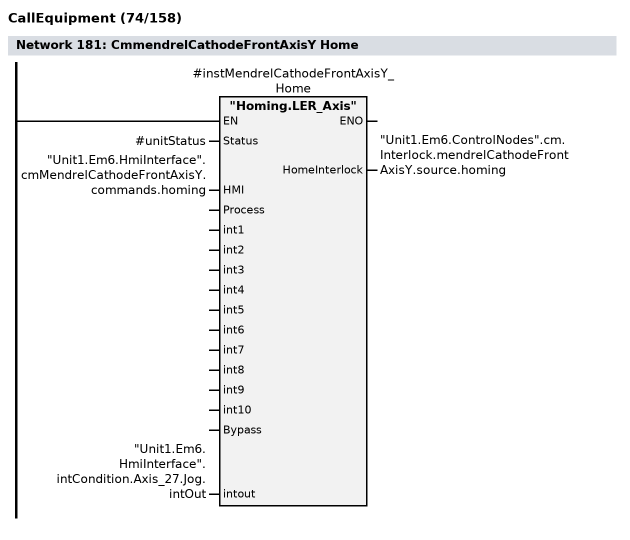
   RUNG wire#powerrail
      #instMendrelCathodeFrontAxisY_Home(Status := #unitStatus, HMI := "Unit1.Em6.HmiInterface".cmMendrelCathodeFrontAxisY.commands.homing, Process :=, int1 :=, int2 :=, int3 :=, int4 :=, int5 :=, int6 :=, int7 :=, int8 :=, int9 :=, int10 :=, Bypass :=, intout := "Unit1.Em6.HmiInterface".intCondition.Axis_27.Jog.intOut, HomeInterlock => "Unit1.Em6.ControlNodes".cm.Interlock.mendrelCathodeFrontAxisY.source.homing)
   END_RUNG
   // the same network as SCL:
   #instMendrelCathodeFrontAxisY_Home(Status := #unitStatus,   // "Homing.LER_Axis"
                           HMI := "Unit1.Em6.HmiInterface".cmMendrelCathodeFrontAxisY.commands.homing,
                           intout := "Unit1.Em6.HmiInterface".intCondition.Axis_27.Jog.intOut,
                           HomeInterlock => "Unit1.Em6.ControlNodes".cm.Interlock.mendrelCathodeFrontAxisY.source.homing);
END_REGION

REGION Network 182: CmMendrelCathodeFrontAxisY Position Absolute Jog
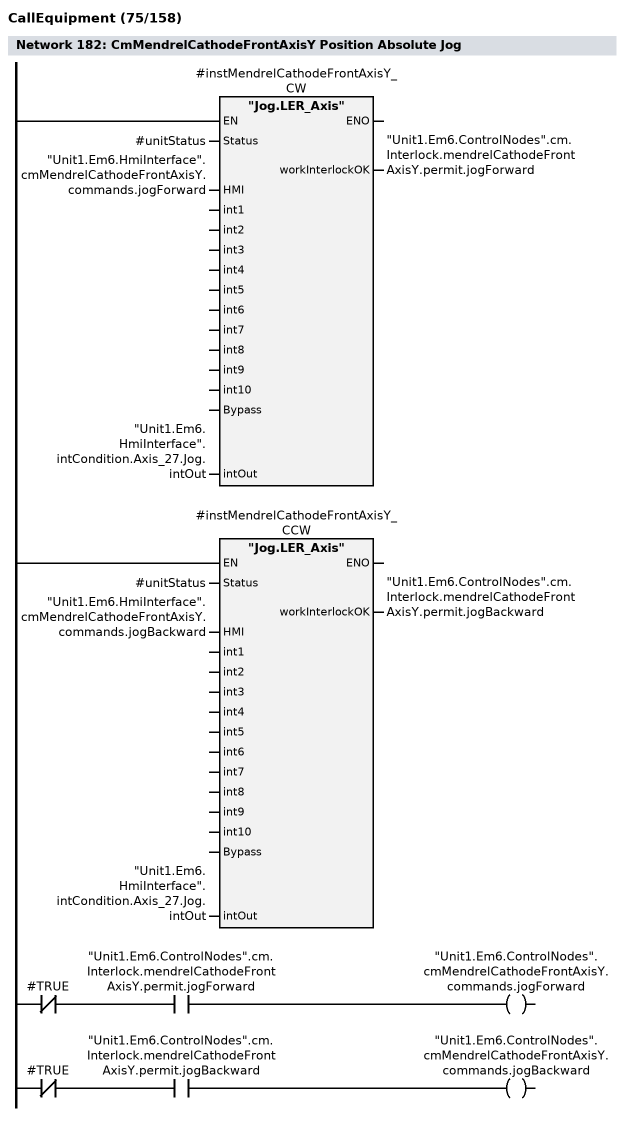
   RUNG wire#powerrail
      #instMendrelCathodeFrontAxisY_CW(Status := #unitStatus, HMI := "Unit1.Em6.HmiInterface".cmMendrelCathodeFrontAxisY.commands.jogForward, int1 :=, int2 :=, int3 :=, int4 :=, int5 :=, int6 :=, int7 :=, int8 :=, int9 :=, int10 :=, Bypass :=, intOut := "Unit1.Em6.HmiInterface".intCondition.Axis_27.Jog.intOut, workInterlockOK => "Unit1.Em6.ControlNodes".cm.Interlock.mendrelCathodeFrontAxisY.permit.jogForward)
   END_RUNG
   RUNG wire#powerrail
      #instMendrelCathodeFrontAxisY_CCW(Status := #unitStatus, HMI := "Unit1.Em6.HmiInterface".cmMendrelCathodeFrontAxisY.commands.jogBackward, int1 :=, int2 :=, int3 :=, int4 :=, int5 :=, int6 :=, int7 :=, int8 :=, int9 :=, int10 :=, Bypass :=, intOut := "Unit1.Em6.HmiInterface".intCondition.Axis_27.Jog.intOut, workInterlockOK => "Unit1.Em6.ControlNodes".cm.Interlock.mendrelCathodeFrontAxisY.permit.jogBackward)
   END_RUNG
   RUNG wire#powerrail
      I_Contact( #TRUE )
      Contact( "Unit1.Em6.ControlNodes".cm.Interlock.mendrelCathodeFrontAxisY.permit.jogForward )
      Coil( "Unit1.Em6.ControlNodes".cmMendrelCathodeFrontAxisY.commands.jogForward )
   END_RUNG
   RUNG wire#powerrail
      I_Contact( #TRUE )
      Contact( "Unit1.Em6.ControlNodes".cm.Interlock.mendrelCathodeFrontAxisY.permit.jogBackward )
      Coil( "Unit1.Em6.ControlNodes".cmMendrelCathodeFrontAxisY.commands.jogBackward )
   END_RUNG
   // the same network as SCL:
   #instMendrelCathodeFrontAxisY_CW(Status := #unitStatus,   // "Jog.LER_Axis"
                           HMI := "Unit1.Em6.HmiInterface".cmMendrelCathodeFrontAxisY.commands.jogForward,
                           intOut := "Unit1.Em6.HmiInterface".intCondition.Axis_27.Jog.intOut,
                           workInterlockOK => "Unit1.Em6.ControlNodes".cm.Interlock.mendrelCathodeFrontAxisY.permit.jogForward);
   #instMendrelCathodeFrontAxisY_CCW(Status := #unitStatus,   // "Jog.LER_Axis"
                           HMI := "Unit1.Em6.HmiInterface".cmMendrelCathodeFrontAxisY.commands.jogBackward,
                           intOut := "Unit1.Em6.HmiInterface".intCondition.Axis_27.Jog.intOut,
                           workInterlockOK => "Unit1.Em6.ControlNodes".cm.Interlock.mendrelCathodeFrontAxisY.permit.jogBackward);
   "Unit1.Em6.ControlNodes".cmMendrelCathodeFrontAxisY.commands.jogForward := NOT #TRUE AND "Unit1.Em6.ControlNodes".cm.Interlock.mendrelCathodeFrontAxisY.permit.jogForward;
   "Unit1.Em6.ControlNodes".cmMendrelCathodeFrontAxisY.commands.jogBackward := NOT #TRUE AND "Unit1.Em6.ControlNodes".cm.Interlock.mendrelCathodeFrontAxisY.permit.jogBackward;
END_REGION

REGION Network 183: CmMendrelCathodeFrontAxisY Position Absolute Position0
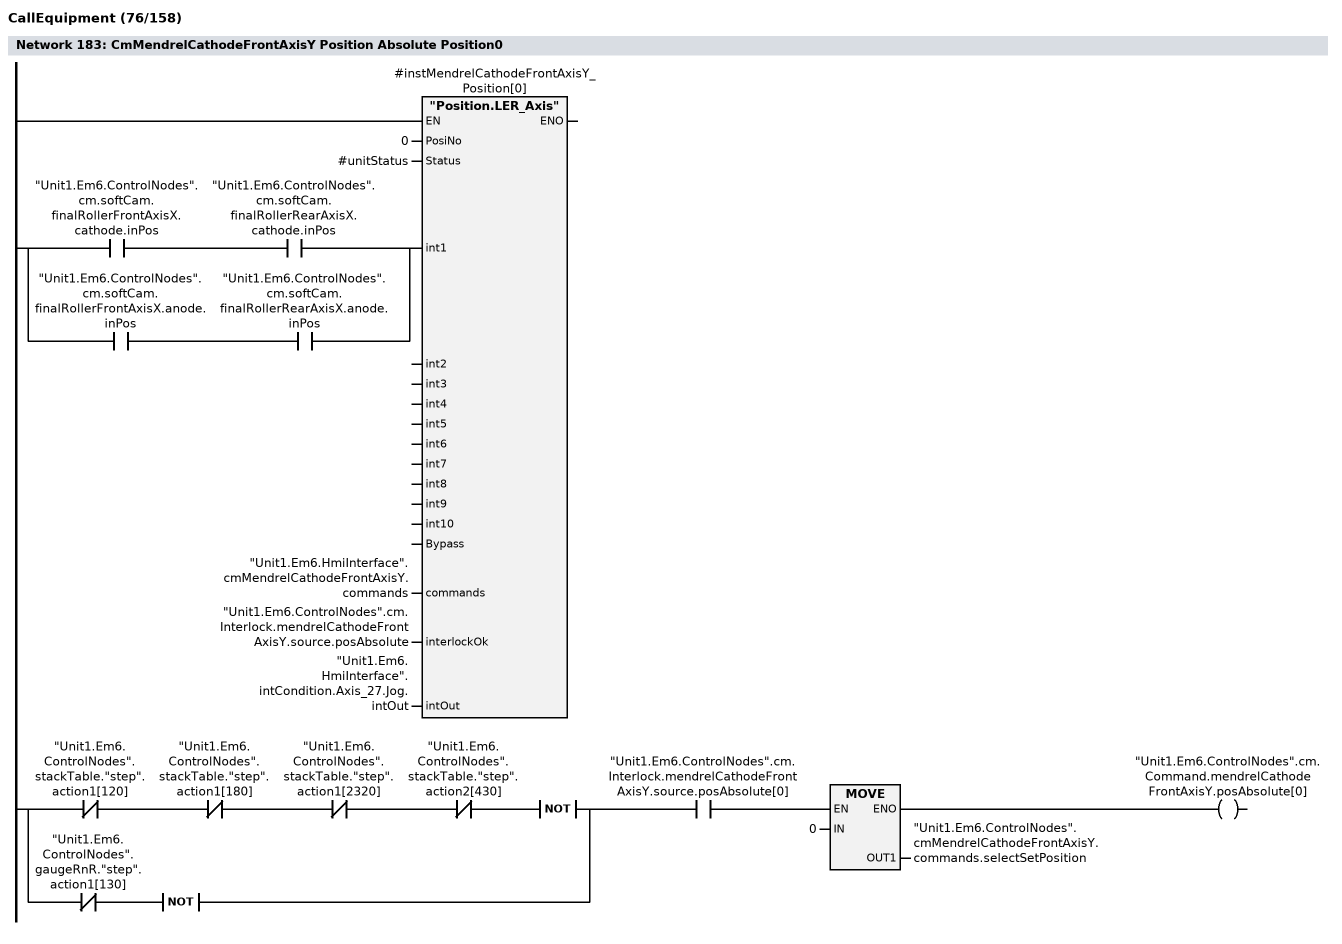
   RUNG wire#powerrail
      #instMendrelCathodeFrontAxisY_Position[0](int1 := wire#w1, PosiNo := 0, Status := #unitStatus, int2 :=, int3 :=, int4 :=, int5 :=, int6 :=, int7 :=, int8 :=, int9 :=, int10 :=, Bypass :=, commands := "Unit1.Em6.HmiInterface".cmMendrelCathodeFrontAxisY.commands, interlockOk := "Unit1.Em6.ControlNodes".cm.Interlock.mendrelCathodeFrontAxisY.source.posAbsolute, intOut := "Unit1.Em6.HmiInterface".intCondition.Axis_27.Jog.intOut)
   END_RUNG
   RUNG wire#powerrail
      Contact( "Unit1.Em6.ControlNodes".cm.softCam.finalRollerFrontAxisX.cathode.inPos )
      Contact( "Unit1.Em6.ControlNodes".cm.softCam.finalRollerRearAxisX.cathode.inPos )
   END_RUNG wire#w1
   RUNG wire#powerrail
      Contact( "Unit1.Em6.ControlNodes".cm.softCam.finalRollerFrontAxisX.anode.inPos )
      Contact( "Unit1.Em6.ControlNodes".cm.softCam.finalRollerRearAxisX.anode.inPos )
   END_RUNG wire#w1
   RUNG wire#powerrail
      I_Contact( "Unit1.Em6.ControlNodes".stackTable."step".action1[120] )
      I_Contact( "Unit1.Em6.ControlNodes".stackTable."step".action1[180] )
      I_Contact( "Unit1.Em6.ControlNodes".stackTable."step".action1[2320] )
      I_Contact( "Unit1.Em6.ControlNodes".stackTable."step".action2[430] )
      Not()
      wire#w2
      Contact( "Unit1.Em6.ControlNodes".cm.Interlock.mendrelCathodeFrontAxisY.source.posAbsolute[0] )
      Move(in := 0, out1 => "Unit1.Em6.ControlNodes".cmMendrelCathodeFrontAxisY.commands.selectSetPosition)
      Coil( "Unit1.Em6.ControlNodes".cm.Command.mendrelCathodeFrontAxisY.posAbsolute[0] )
   END_RUNG
   RUNG wire#powerrail
      I_Contact( "Unit1.Em6.ControlNodes".gaugeRnR."step".action1[130] )
      Not()
   END_RUNG wire#w2
   // the same network as SCL:
   #instMendrelCathodeFrontAxisY_Position[0](PosiNo := 0,   // "Position.LER_Axis"
                           Status := #unitStatus,
                           int1 := ("Unit1.Em6.ControlNodes".cm.softCam.finalRollerFrontAxisX.cathode.inPos AND "Unit1.Em6.ControlNodes".cm.softCam.finalRollerRearAxisX.cathode.inPos) OR ("Unit1.Em6.ControlNodes".cm.softCam.finalRollerFrontAxisX.anode.inPos AND "Unit1.Em6.ControlNodes".cm.softCam.finalRollerRearAxisX.anode.inPos),
                           commands := "Unit1.Em6.HmiInterface".cmMendrelCathodeFrontAxisY.commands,
                           interlockOk := "Unit1.Em6.ControlNodes".cm.Interlock.mendrelCathodeFrontAxisY.source.posAbsolute,
                           intOut := "Unit1.Em6.HmiInterface".intCondition.Axis_27.Jog.intOut);
   #_w1 := (NOT (NOT "Unit1.Em6.ControlNodes".stackTable."step".action1[120] AND NOT "Unit1.Em6.ControlNodes".stackTable."step".action1[180] AND NOT "Unit1.Em6.ControlNodes".stackTable."step".action1[2320] AND NOT "Unit1.Em6.ControlNodes".stackTable."step".action2[430]) OR NOT (NOT "Unit1.Em6.ControlNodes".gaugeRnR."step".action1[130])) AND "Unit1.Em6.ControlNodes".cm.Interlock.mendrelCathodeFrontAxisY.source.posAbsolute[0];
   IF #_w1 THEN "Unit1.Em6.ControlNodes".cmMendrelCathodeFrontAxisY.commands.selectSetPosition := 0; END_IF;
   "Unit1.Em6.ControlNodes".cm.Command.mendrelCathodeFrontAxisY.posAbsolute[0] := #_w1;
END_REGION

REGION Network 184: CmMendrelCathodeFrontAxisY Position Absolute Position1
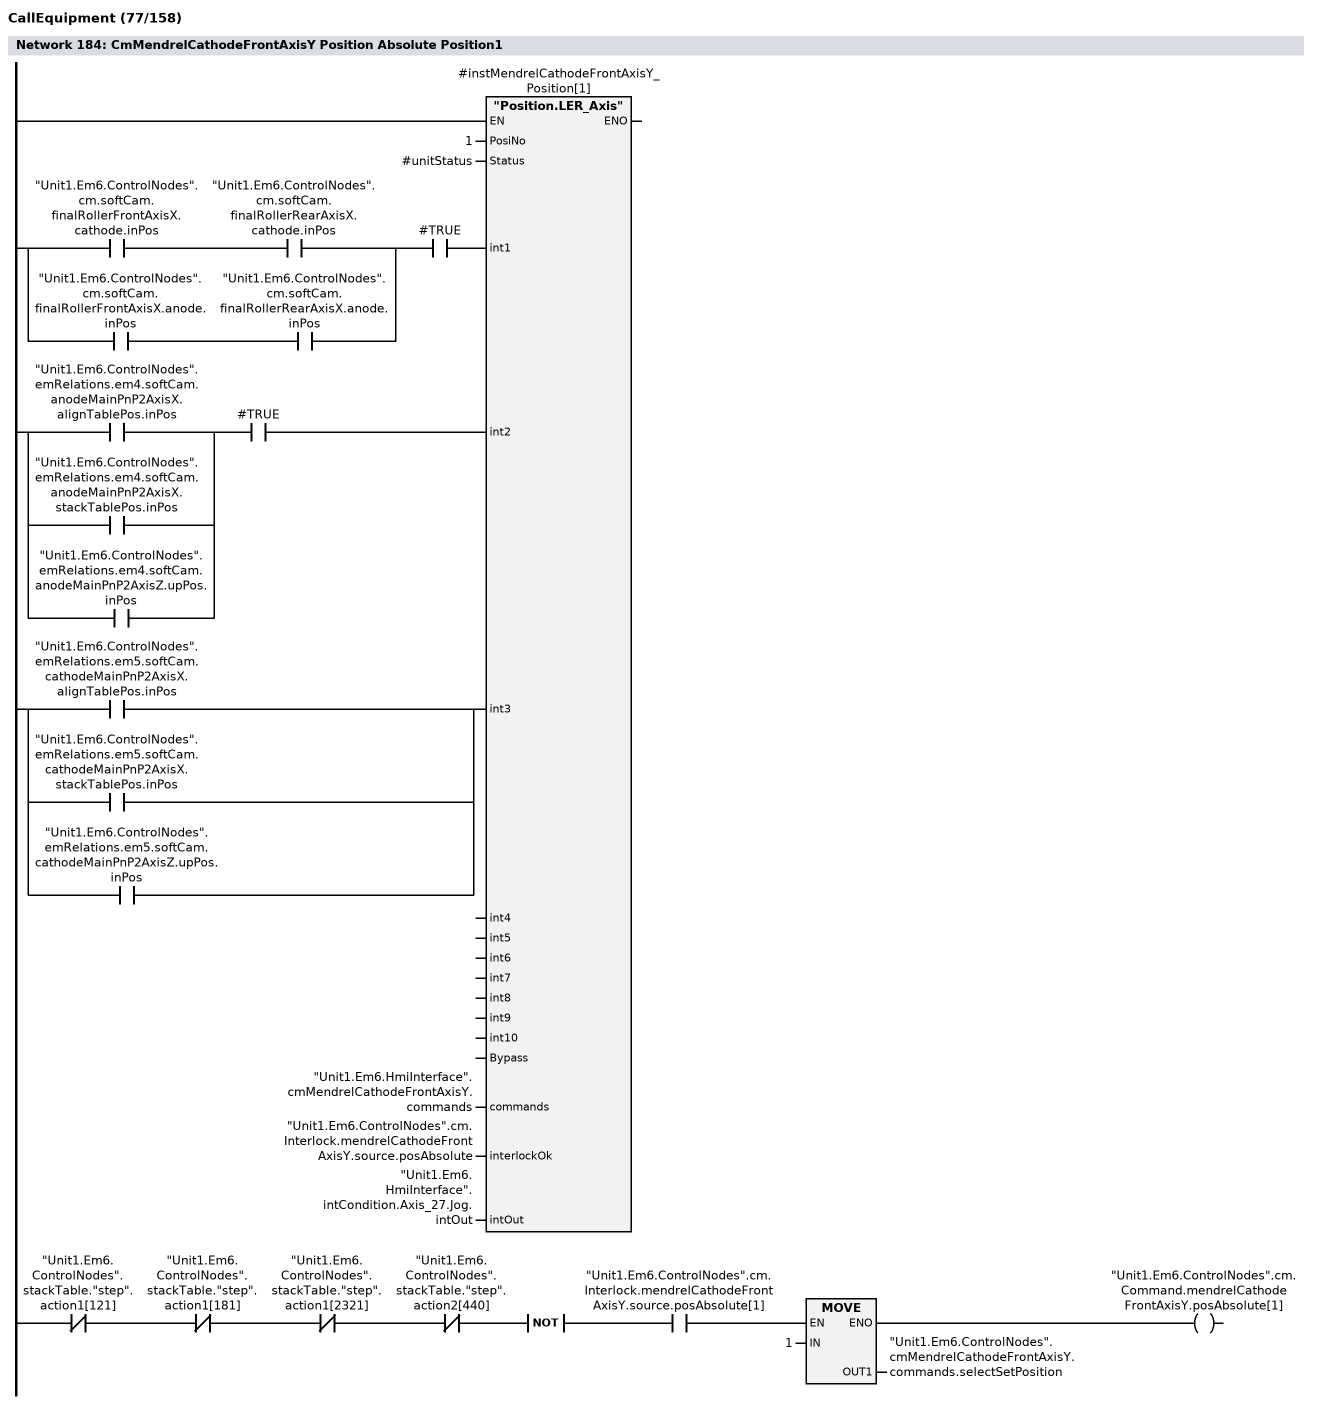
   RUNG wire#powerrail
      #instMendrelCathodeFrontAxisY_Position[1](int1 := wire#w2, int2 := wire#w4, int3 := wire#w5, PosiNo := 1, Status := #unitStatus, int4 :=, int5 :=, int6 :=, int7 :=, int8 :=, int9 :=, int10 :=, Bypass :=, commands := "Unit1.Em6.HmiInterface".cmMendrelCathodeFrontAxisY.commands, interlockOk := "Unit1.Em6.ControlNodes".cm.Interlock.mendrelCathodeFrontAxisY.source.posAbsolute, intOut := "Unit1.Em6.HmiInterface".intCondition.Axis_27.Jog.intOut)
   END_RUNG
   RUNG wire#powerrail
      Contact( "Unit1.Em6.ControlNodes".cm.softCam.finalRollerFrontAxisX.cathode.inPos )
      Contact( "Unit1.Em6.ControlNodes".cm.softCam.finalRollerRearAxisX.cathode.inPos )
      wire#w1
      Contact( #TRUE )
   END_RUNG wire#w2
   RUNG wire#powerrail
      Contact( "Unit1.Em6.ControlNodes".cm.softCam.finalRollerFrontAxisX.anode.inPos )
      Contact( "Unit1.Em6.ControlNodes".cm.softCam.finalRollerRearAxisX.anode.inPos )
   END_RUNG wire#w1
   RUNG wire#powerrail
      Contact( "Unit1.Em6.ControlNodes".emRelations.em4.softCam.anodeMainPnP2AxisX.alignTablePos.inPos )
      wire#w3
      Contact( #TRUE )
   END_RUNG wire#w4
   RUNG wire#powerrail
      Contact( "Unit1.Em6.ControlNodes".emRelations.em4.softCam.anodeMainPnP2AxisX.stackTablePos.inPos )
   END_RUNG wire#w3
   RUNG wire#powerrail
      Contact( "Unit1.Em6.ControlNodes".emRelations.em4.softCam.anodeMainPnP2AxisZ.upPos.inPos )
   END_RUNG wire#w3
   RUNG wire#powerrail
      Contact( "Unit1.Em6.ControlNodes".emRelations.em5.softCam.cathodeMainPnP2AxisX.alignTablePos.inPos )
   END_RUNG wire#w5
   RUNG wire#powerrail
      Contact( "Unit1.Em6.ControlNodes".emRelations.em5.softCam.cathodeMainPnP2AxisX.stackTablePos.inPos )
   END_RUNG wire#w5
   RUNG wire#powerrail
      Contact( "Unit1.Em6.ControlNodes".emRelations.em5.softCam.cathodeMainPnP2AxisZ.upPos.inPos )
   END_RUNG wire#w5
   RUNG wire#powerrail
      I_Contact( "Unit1.Em6.ControlNodes".stackTable."step".action1[121] )
      I_Contact( "Unit1.Em6.ControlNodes".stackTable."step".action1[181] )
      I_Contact( "Unit1.Em6.ControlNodes".stackTable."step".action1[2321] )
      I_Contact( "Unit1.Em6.ControlNodes".stackTable."step".action2[440] )
      Not()
      Contact( "Unit1.Em6.ControlNodes".cm.Interlock.mendrelCathodeFrontAxisY.source.posAbsolute[1] )
      Move(in := 1, out1 => "Unit1.Em6.ControlNodes".cmMendrelCathodeFrontAxisY.commands.selectSetPosition)
      Coil( "Unit1.Em6.ControlNodes".cm.Command.mendrelCathodeFrontAxisY.posAbsolute[1] )
   END_RUNG
   // the same network as SCL:
   #instMendrelCathodeFrontAxisY_Position[1](PosiNo := 1,   // "Position.LER_Axis"
                           Status := #unitStatus,
                           int1 := (("Unit1.Em6.ControlNodes".cm.softCam.finalRollerFrontAxisX.cathode.inPos AND "Unit1.Em6.ControlNodes".cm.softCam.finalRollerRearAxisX.cathode.inPos) OR ("Unit1.Em6.ControlNodes".cm.softCam.finalRollerFrontAxisX.anode.inPos AND "Unit1.Em6.ControlNodes".cm.softCam.finalRollerRearAxisX.anode.inPos)) AND #TRUE,
                           int2 := ("Unit1.Em6.ControlNodes".emRelations.em4.softCam.anodeMainPnP2AxisX.alignTablePos.inPos OR "Unit1.Em6.ControlNodes".emRelations.em4.softCam.anodeMainPnP2AxisX.stackTablePos.inPos OR "Unit1.Em6.ControlNodes".emRelations.em4.softCam.anodeMainPnP2AxisZ.upPos.inPos) AND #TRUE,
                           int3 := "Unit1.Em6.ControlNodes".emRelations.em5.softCam.cathodeMainPnP2AxisX.alignTablePos.inPos OR "Unit1.Em6.ControlNodes".emRelations.em5.softCam.cathodeMainPnP2AxisX.stackTablePos.inPos OR "Unit1.Em6.ControlNodes".emRelations.em5.softCam.cathodeMainPnP2AxisZ.upPos.inPos,
                           commands := "Unit1.Em6.HmiInterface".cmMendrelCathodeFrontAxisY.commands,
                           interlockOk := "Unit1.Em6.ControlNodes".cm.Interlock.mendrelCathodeFrontAxisY.source.posAbsolute,
                           intOut := "Unit1.Em6.HmiInterface".intCondition.Axis_27.Jog.intOut);
   #_w1 := NOT (NOT "Unit1.Em6.ControlNodes".stackTable."step".action1[121] AND NOT "Unit1.Em6.ControlNodes".stackTable."step".action1[181] AND NOT "Unit1.Em6.ControlNodes".stackTable."step".action1[2321] AND NOT "Unit1.Em6.ControlNodes".stackTable."step".action2[440]) AND "Unit1.Em6.ControlNodes".cm.Interlock.mendrelCathodeFrontAxisY.source.posAbsolute[1];
   IF #_w1 THEN "Unit1.Em6.ControlNodes".cmMendrelCathodeFrontAxisY.commands.selectSetPosition := 1; END_IF;
   "Unit1.Em6.ControlNodes".cm.Command.mendrelCathodeFrontAxisY.posAbsolute[1] := #_w1;
END_REGION

REGION Network 185: CmMendrelCathodeFrontAxisY Position Absolute Position2
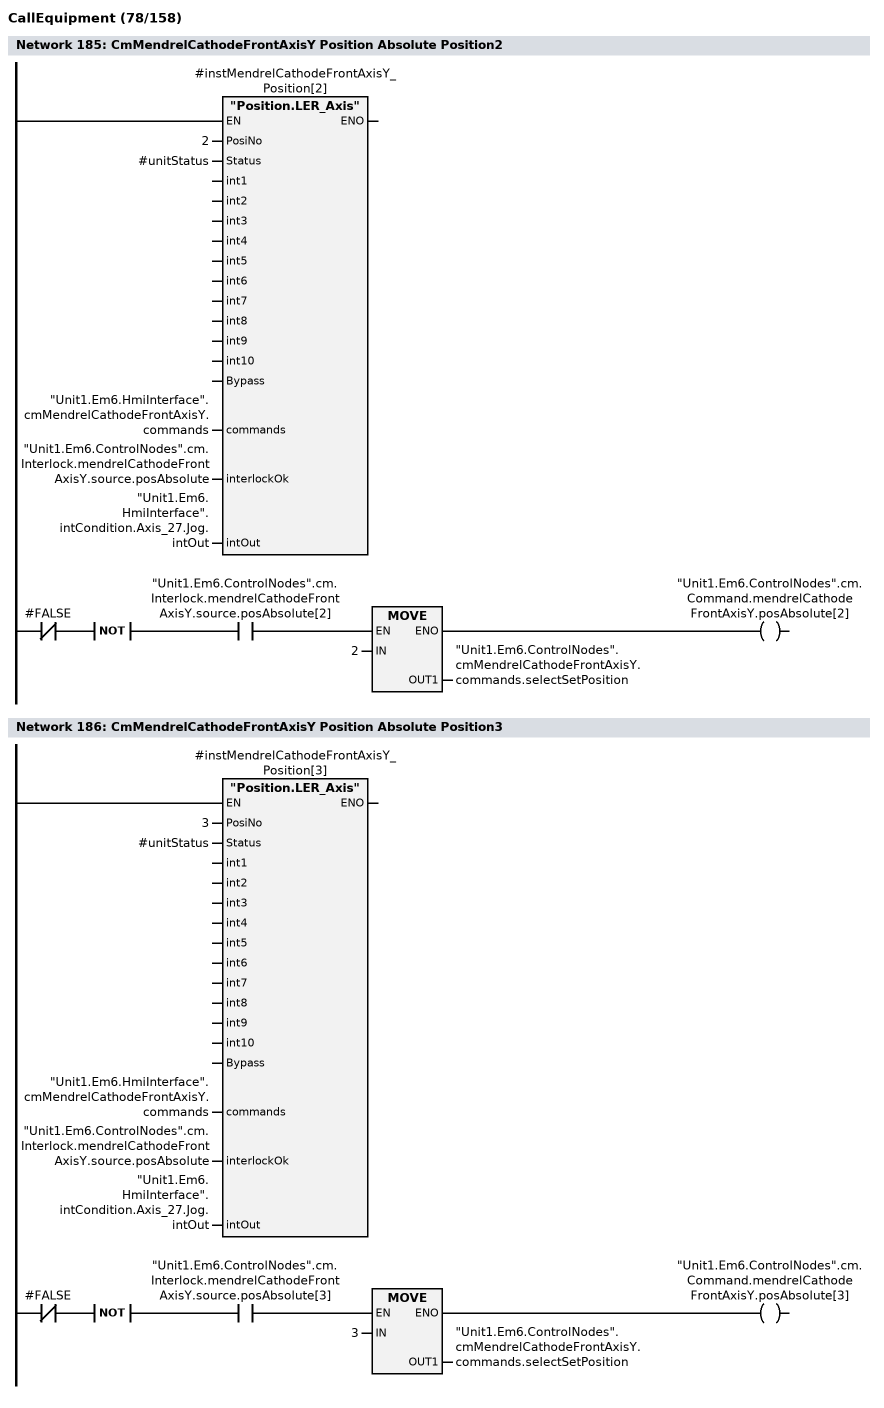
   RUNG wire#powerrail
      #instMendrelCathodeFrontAxisY_Position[2](PosiNo := 2, Status := #unitStatus, int1 :=, int2 :=, int3 :=, int4 :=, int5 :=, int6 :=, int7 :=, int8 :=, int9 :=, int10 :=, Bypass :=, commands := "Unit1.Em6.HmiInterface".cmMendrelCathodeFrontAxisY.commands, interlockOk := "Unit1.Em6.ControlNodes".cm.Interlock.mendrelCathodeFrontAxisY.source.posAbsolute, intOut := "Unit1.Em6.HmiInterface".intCondition.Axis_27.Jog.intOut)
   END_RUNG
   RUNG wire#powerrail
      I_Contact( #FALSE )
      Not()
      Contact( "Unit1.Em6.ControlNodes".cm.Interlock.mendrelCathodeFrontAxisY.source.posAbsolute[2] )
      Move(in := 2, out1 => "Unit1.Em6.ControlNodes".cmMendrelCathodeFrontAxisY.commands.selectSetPosition)
      Coil( "Unit1.Em6.ControlNodes".cm.Command.mendrelCathodeFrontAxisY.posAbsolute[2] )
   END_RUNG
   // the same network as SCL:
   #instMendrelCathodeFrontAxisY_Position[2](PosiNo := 2,   // "Position.LER_Axis"
                           Status := #unitStatus,
                           commands := "Unit1.Em6.HmiInterface".cmMendrelCathodeFrontAxisY.commands,
                           interlockOk := "Unit1.Em6.ControlNodes".cm.Interlock.mendrelCathodeFrontAxisY.source.posAbsolute,
                           intOut := "Unit1.Em6.HmiInterface".intCondition.Axis_27.Jog.intOut);
   #_w1 := NOT (NOT #FALSE) AND "Unit1.Em6.ControlNodes".cm.Interlock.mendrelCathodeFrontAxisY.source.posAbsolute[2];
   IF #_w1 THEN "Unit1.Em6.ControlNodes".cmMendrelCathodeFrontAxisY.commands.selectSetPosition := 2; END_IF;
   "Unit1.Em6.ControlNodes".cm.Command.mendrelCathodeFrontAxisY.posAbsolute[2] := #_w1;
END_REGION

REGION Network 186: CmMendrelCathodeFrontAxisY Position Absolute Position3
   RUNG wire#powerrail
      #instMendrelCathodeFrontAxisY_Position[3](PosiNo := 3, Status := #unitStatus, int1 :=, int2 :=, int3 :=, int4 :=, int5 :=, int6 :=, int7 :=, int8 :=, int9 :=, int10 :=, Bypass :=, commands := "Unit1.Em6.HmiInterface".cmMendrelCathodeFrontAxisY.commands, interlockOk := "Unit1.Em6.ControlNodes".cm.Interlock.mendrelCathodeFrontAxisY.source.posAbsolute, intOut := "Unit1.Em6.HmiInterface".intCondition.Axis_27.Jog.intOut)
   END_RUNG
   RUNG wire#powerrail
      I_Contact( #FALSE )
      Not()
      Contact( "Unit1.Em6.ControlNodes".cm.Interlock.mendrelCathodeFrontAxisY.source.posAbsolute[3] )
      Move(in := 3, out1 => "Unit1.Em6.ControlNodes".cmMendrelCathodeFrontAxisY.commands.selectSetPosition)
      Coil( "Unit1.Em6.ControlNodes".cm.Command.mendrelCathodeFrontAxisY.posAbsolute[3] )
   END_RUNG
   // the same network as SCL:
   #instMendrelCathodeFrontAxisY_Position[3](PosiNo := 3,   // "Position.LER_Axis"
                           Status := #unitStatus,
                           commands := "Unit1.Em6.HmiInterface".cmMendrelCathodeFrontAxisY.commands,
                           interlockOk := "Unit1.Em6.ControlNodes".cm.Interlock.mendrelCathodeFrontAxisY.source.posAbsolute,
                           intOut := "Unit1.Em6.HmiInterface".intCondition.Axis_27.Jog.intOut);
   #_w1 := NOT (NOT #FALSE) AND "Unit1.Em6.ControlNodes".cm.Interlock.mendrelCathodeFrontAxisY.source.posAbsolute[3];
   IF #_w1 THEN "Unit1.Em6.ControlNodes".cmMendrelCathodeFrontAxisY.commands.selectSetPosition := 3; END_IF;
   "Unit1.Em6.ControlNodes".cm.Command.mendrelCathodeFrontAxisY.posAbsolute[3] := #_w1;
END_REGION

REGION Network 187: CmMendrelCathodeFrontAxisY Position Absolute Position4
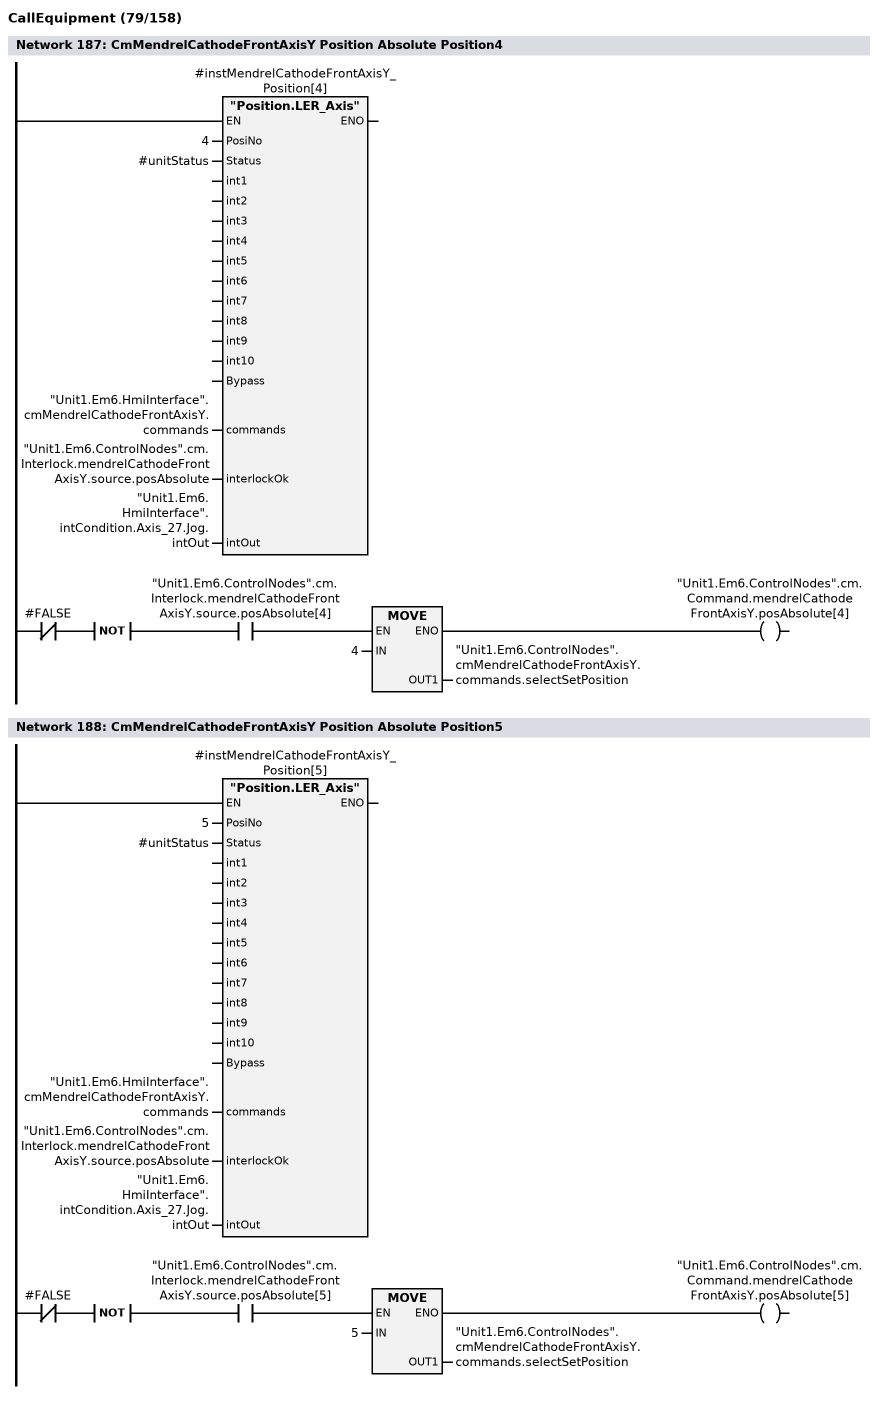
   RUNG wire#powerrail
      #instMendrelCathodeFrontAxisY_Position[4](PosiNo := 4, Status := #unitStatus, int1 :=, int2 :=, int3 :=, int4 :=, int5 :=, int6 :=, int7 :=, int8 :=, int9 :=, int10 :=, Bypass :=, commands := "Unit1.Em6.HmiInterface".cmMendrelCathodeFrontAxisY.commands, interlockOk := "Unit1.Em6.ControlNodes".cm.Interlock.mendrelCathodeFrontAxisY.source.posAbsolute, intOut := "Unit1.Em6.HmiInterface".intCondition.Axis_27.Jog.intOut)
   END_RUNG
   RUNG wire#powerrail
      I_Contact( #FALSE )
      Not()
      Contact( "Unit1.Em6.ControlNodes".cm.Interlock.mendrelCathodeFrontAxisY.source.posAbsolute[4] )
      Move(in := 4, out1 => "Unit1.Em6.ControlNodes".cmMendrelCathodeFrontAxisY.commands.selectSetPosition)
      Coil( "Unit1.Em6.ControlNodes".cm.Command.mendrelCathodeFrontAxisY.posAbsolute[4] )
   END_RUNG
   // the same network as SCL:
   #instMendrelCathodeFrontAxisY_Position[4](PosiNo := 4,   // "Position.LER_Axis"
                           Status := #unitStatus,
                           commands := "Unit1.Em6.HmiInterface".cmMendrelCathodeFrontAxisY.commands,
                           interlockOk := "Unit1.Em6.ControlNodes".cm.Interlock.mendrelCathodeFrontAxisY.source.posAbsolute,
                           intOut := "Unit1.Em6.HmiInterface".intCondition.Axis_27.Jog.intOut);
   #_w1 := NOT (NOT #FALSE) AND "Unit1.Em6.ControlNodes".cm.Interlock.mendrelCathodeFrontAxisY.source.posAbsolute[4];
   IF #_w1 THEN "Unit1.Em6.ControlNodes".cmMendrelCathodeFrontAxisY.commands.selectSetPosition := 4; END_IF;
   "Unit1.Em6.ControlNodes".cm.Command.mendrelCathodeFrontAxisY.posAbsolute[4] := #_w1;
END_REGION

REGION Network 188: CmMendrelCathodeFrontAxisY Position Absolute Position5
   RUNG wire#powerrail
      #instMendrelCathodeFrontAxisY_Position[5](PosiNo := 5, Status := #unitStatus, int1 :=, int2 :=, int3 :=, int4 :=, int5 :=, int6 :=, int7 :=, int8 :=, int9 :=, int10 :=, Bypass :=, commands := "Unit1.Em6.HmiInterface".cmMendrelCathodeFrontAxisY.commands, interlockOk := "Unit1.Em6.ControlNodes".cm.Interlock.mendrelCathodeFrontAxisY.source.posAbsolute, intOut := "Unit1.Em6.HmiInterface".intCondition.Axis_27.Jog.intOut)
   END_RUNG
   RUNG wire#powerrail
      I_Contact( #FALSE )
      Not()
      Contact( "Unit1.Em6.ControlNodes".cm.Interlock.mendrelCathodeFrontAxisY.source.posAbsolute[5] )
      Move(in := 5, out1 => "Unit1.Em6.ControlNodes".cmMendrelCathodeFrontAxisY.commands.selectSetPosition)
      Coil( "Unit1.Em6.ControlNodes".cm.Command.mendrelCathodeFrontAxisY.posAbsolute[5] )
   END_RUNG
   // the same network as SCL:
   #instMendrelCathodeFrontAxisY_Position[5](PosiNo := 5,   // "Position.LER_Axis"
                           Status := #unitStatus,
                           commands := "Unit1.Em6.HmiInterface".cmMendrelCathodeFrontAxisY.commands,
                           interlockOk := "Unit1.Em6.ControlNodes".cm.Interlock.mendrelCathodeFrontAxisY.source.posAbsolute,
                           intOut := "Unit1.Em6.HmiInterface".intCondition.Axis_27.Jog.intOut);
   #_w1 := NOT (NOT #FALSE) AND "Unit1.Em6.ControlNodes".cm.Interlock.mendrelCathodeFrontAxisY.source.posAbsolute[5];
   IF #_w1 THEN "Unit1.Em6.ControlNodes".cmMendrelCathodeFrontAxisY.commands.selectSetPosition := 5; END_IF;
   "Unit1.Em6.ControlNodes".cm.Command.mendrelCathodeFrontAxisY.posAbsolute[5] := #_w1;
END_REGION

REGION Network 189: CmMendrelCathodeFrontAxisY Summary Command
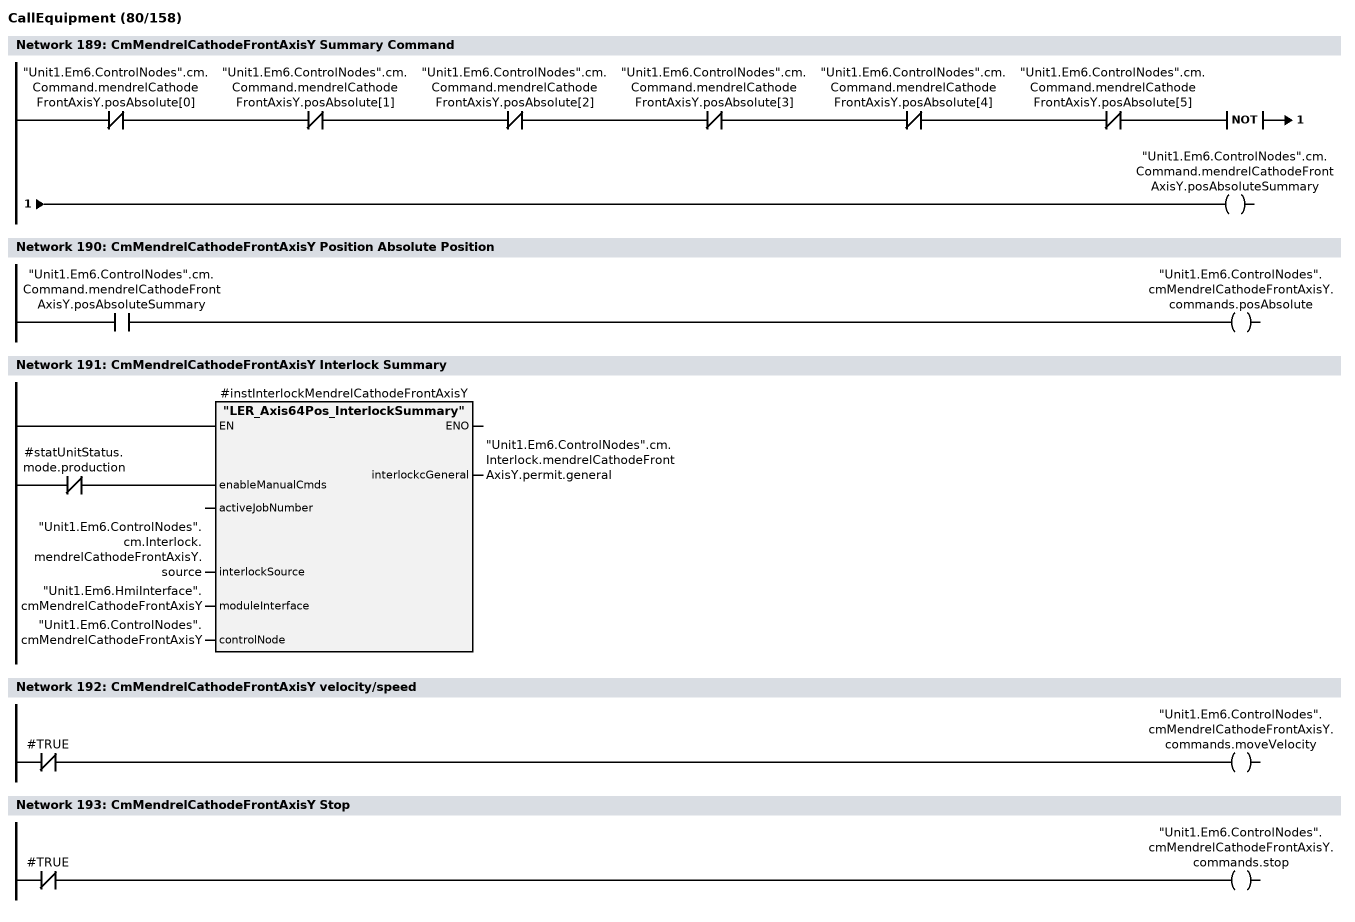
   RUNG wire#powerrail
      I_Contact( "Unit1.Em6.ControlNodes".cm.Command.mendrelCathodeFrontAxisY.posAbsolute[0] )
      I_Contact( "Unit1.Em6.ControlNodes".cm.Command.mendrelCathodeFrontAxisY.posAbsolute[1] )
      I_Contact( "Unit1.Em6.ControlNodes".cm.Command.mendrelCathodeFrontAxisY.posAbsolute[2] )
      I_Contact( "Unit1.Em6.ControlNodes".cm.Command.mendrelCathodeFrontAxisY.posAbsolute[3] )
      I_Contact( "Unit1.Em6.ControlNodes".cm.Command.mendrelCathodeFrontAxisY.posAbsolute[4] )
      I_Contact( "Unit1.Em6.ControlNodes".cm.Command.mendrelCathodeFrontAxisY.posAbsolute[5] )
      Not()
      Coil( "Unit1.Em6.ControlNodes".cm.Command.mendrelCathodeFrontAxisY.posAbsoluteSummary )
   END_RUNG
   // the same network as SCL:
   "Unit1.Em6.ControlNodes".cm.Command.mendrelCathodeFrontAxisY.posAbsoluteSummary := NOT (NOT "Unit1.Em6.ControlNodes".cm.Command.mendrelCathodeFrontAxisY.posAbsolute[0] AND NOT "Unit1.Em6.ControlNodes".cm.Command.mendrelCathodeFrontAxisY.posAbsolute[1] AND NOT "Unit1.Em6.ControlNodes".cm.Command.mendrelCathodeFrontAxisY.posAbsolute[2] AND NOT "Unit1.Em6.ControlNodes".cm.Command.mendrelCathodeFrontAxisY.posAbsolute[3] AND NOT "Unit1.Em6.ControlNodes".cm.Command.mendrelCathodeFrontAxisY.posAbsolute[4] AND NOT "Unit1.Em6.ControlNodes".cm.Command.mendrelCathodeFrontAxisY.posAbsolute[5]);
END_REGION

REGION Network 190: CmMendrelCathodeFrontAxisY Position Absolute Position
   RUNG wire#powerrail
      Contact( "Unit1.Em6.ControlNodes".cm.Command.mendrelCathodeFrontAxisY.posAbsoluteSummary )
      Coil( "Unit1.Em6.ControlNodes".cmMendrelCathodeFrontAxisY.commands.posAbsolute )
   END_RUNG
   // the same network as SCL:
   "Unit1.Em6.ControlNodes".cmMendrelCathodeFrontAxisY.commands.posAbsolute := "Unit1.Em6.ControlNodes".cm.Command.mendrelCathodeFrontAxisY.posAbsoluteSummary;
END_REGION

REGION Network 191: CmMendrelCathodeFrontAxisY Interlock Summary
   RUNG wire#powerrail
      #instInterlockMendrelCathodeFrontAxisY(enableManualCmds := wire#w1, activeJobNumber :=, interlockSource := "Unit1.Em6.ControlNodes".cm.Interlock.mendrelCathodeFrontAxisY.source, moduleInterface := "Unit1.Em6.HmiInterface".cmMendrelCathodeFrontAxisY, controlNode := "Unit1.Em6.ControlNodes".cmMendrelCathodeFrontAxisY, interlockcGeneral => "Unit1.Em6.ControlNodes".cm.Interlock.mendrelCathodeFrontAxisY.permit.general)
   END_RUNG
   RUNG wire#powerrail
      I_Contact( #statUnitStatus.mode.production )
   END_RUNG wire#w1
   // the same network as SCL:
   #instInterlockMendrelCathodeFrontAxisY(enableManualCmds := NOT #statUnitStatus.mode.production,   // "LER_Axis64Pos_InterlockSummary"
                           interlockSource := "Unit1.Em6.ControlNodes".cm.Interlock.mendrelCathodeFrontAxisY.source,
                           moduleInterface := "Unit1.Em6.HmiInterface".cmMendrelCathodeFrontAxisY,
                           controlNode := "Unit1.Em6.ControlNodes".cmMendrelCathodeFrontAxisY,
                           interlockcGeneral => "Unit1.Em6.ControlNodes".cm.Interlock.mendrelCathodeFrontAxisY.permit.general);
END_REGION

REGION Network 192: CmMendrelCathodeFrontAxisY velocity/speed
   RUNG wire#powerrail
      I_Contact( #TRUE )
      Coil( "Unit1.Em6.ControlNodes".cmMendrelCathodeFrontAxisY.commands.moveVelocity )
   END_RUNG
   // the same network as SCL:
   "Unit1.Em6.ControlNodes".cmMendrelCathodeFrontAxisY.commands.moveVelocity := NOT #TRUE;
END_REGION

REGION Network 193: CmMendrelCathodeFrontAxisY Stop
   RUNG wire#powerrail
      I_Contact( #TRUE )
      Coil( "Unit1.Em6.ControlNodes".cmMendrelCathodeFrontAxisY.commands.stop )
   END_RUNG
   // the same network as SCL:
   "Unit1.Em6.ControlNodes".cmMendrelCathodeFrontAxisY.commands.stop := NOT #TRUE;
END_REGION

REGION Network 194: Call CM Cathode Mandrel Front Y-Axis (LBC_Axis64Pos)
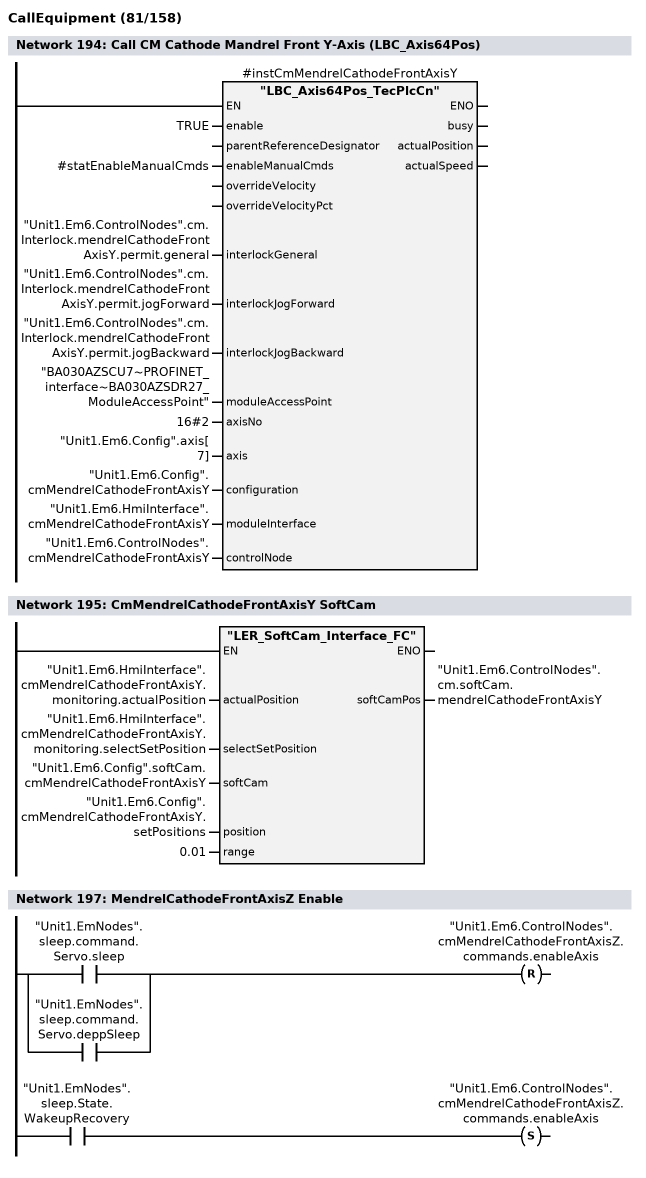
   RUNG wire#powerrail
      #instCmMendrelCathodeFrontAxisY(enable := TRUE, parentReferenceDesignator :=, enableManualCmds := #statEnableManualCmds, overrideVelocity :=, overrideVelocityPct :=, interlockGeneral := "Unit1.Em6.ControlNodes".cm.Interlock.mendrelCathodeFrontAxisY.permit.general, interlockJogForward := "Unit1.Em6.ControlNodes".cm.Interlock.mendrelCathodeFrontAxisY.permit.jogForward, interlockJogBackward := "Unit1.Em6.ControlNodes".cm.Interlock.mendrelCathodeFrontAxisY.permit.jogBackward, moduleAccessPoint := "BA030AZSCU7~PROFINET_interface~BA030AZSDR27_ModuleAccessPoint", axisNo := 16#2, axis := "Unit1.Em6.Config".axis[7], configuration := "Unit1.Em6.Config".cmMendrelCathodeFrontAxisY, moduleInterface := "Unit1.Em6.HmiInterface".cmMendrelCathodeFrontAxisY, controlNode := "Unit1.Em6.ControlNodes".cmMendrelCathodeFrontAxisY, busy =>, actualPosition =>, actualSpeed =>)
   END_RUNG
   // the same network as SCL:
   #instCmMendrelCathodeFrontAxisY(enable := TRUE,   // "LBC_Axis64Pos_TecPlcCn"
                           enableManualCmds := #statEnableManualCmds,
                           interlockGeneral := "Unit1.Em6.ControlNodes".cm.Interlock.mendrelCathodeFrontAxisY.permit.general,
                           interlockJogForward := "Unit1.Em6.ControlNodes".cm.Interlock.mendrelCathodeFrontAxisY.permit.jogForward,
                           interlockJogBackward := "Unit1.Em6.ControlNodes".cm.Interlock.mendrelCathodeFrontAxisY.permit.jogBackward,
                           moduleAccessPoint := "BA030AZSCU7~PROFINET_interface~BA030AZSDR27_ModuleAccessPoint",
                           axisNo := 16#2,
                           axis := "Unit1.Em6.Config".axis[7],
                           configuration := "Unit1.Em6.Config".cmMendrelCathodeFrontAxisY,
                           moduleInterface := "Unit1.Em6.HmiInterface".cmMendrelCathodeFrontAxisY,
                           controlNode := "Unit1.Em6.ControlNodes".cmMendrelCathodeFrontAxisY);
END_REGION

REGION Network 195: CmMendrelCathodeFrontAxisY SoftCam
   RUNG wire#powerrail
      "LER_SoftCam_Interface_FC"(actualPosition := "Unit1.Em6.HmiInterface".cmMendrelCathodeFrontAxisY.monitoring.actualPosition, selectSetPosition := "Unit1.Em6.HmiInterface".cmMendrelCathodeFrontAxisY.monitoring.selectSetPosition, softCam := "Unit1.Em6.Config".softCam.cmMendrelCathodeFrontAxisY, position := "Unit1.Em6.Config".cmMendrelCathodeFrontAxisY.setPositions, range := 0.01, softCamPos => "Unit1.Em6.ControlNodes".cm.softCam.mendrelCathodeFrontAxisY)
   END_RUNG
   // the same network as SCL:
   "LER_SoftCam_Interface_FC"(actualPosition := "Unit1.Em6.HmiInterface".cmMendrelCathodeFrontAxisY.monitoring.actualPosition,
                           selectSetPosition := "Unit1.Em6.HmiInterface".cmMendrelCathodeFrontAxisY.monitoring.selectSetPosition,
                           softCam := "Unit1.Em6.Config".softCam.cmMendrelCathodeFrontAxisY,
                           position := "Unit1.Em6.Config".cmMendrelCathodeFrontAxisY.setPositions,
                           range := 0.01,
                           softCamPos => "Unit1.Em6.ControlNodes".cm.softCam.mendrelCathodeFrontAxisY);
END_REGION

REGION Network 197: MendrelCathodeFrontAxisZ Enable
   RUNG wire#powerrail
      Contact( "Unit1.EmNodes".sleep.command.Servo.sleep )
      wire#w1
      R_Coil( "Unit1.Em6.ControlNodes".cmMendrelCathodeFrontAxisZ.commands.enableAxis )
   END_RUNG
   RUNG wire#powerrail
      Contact( "Unit1.EmNodes".sleep.command.Servo.deppSleep )
   END_RUNG wire#w1
   RUNG wire#powerrail
      Contact( "Unit1.EmNodes".sleep.State.WakeupRecovery )
      S_Coil( "Unit1.Em6.ControlNodes".cmMendrelCathodeFrontAxisZ.commands.enableAxis )
   END_RUNG
   // the same network as SCL:
   IF "Unit1.EmNodes".sleep.command.Servo.sleep OR "Unit1.EmNodes".sleep.command.Servo.deppSleep THEN
       "Unit1.Em6.ControlNodes".cmMendrelCathodeFrontAxisZ.commands.enableAxis := FALSE;
   END_IF;
   IF "Unit1.EmNodes".sleep.State.WakeupRecovery THEN
       "Unit1.Em6.ControlNodes".cmMendrelCathodeFrontAxisZ.commands.enableAxis := TRUE;
   END_IF;
END_REGION

REGION Network 198: CmmendrelCathodeFrontAxisZ Home
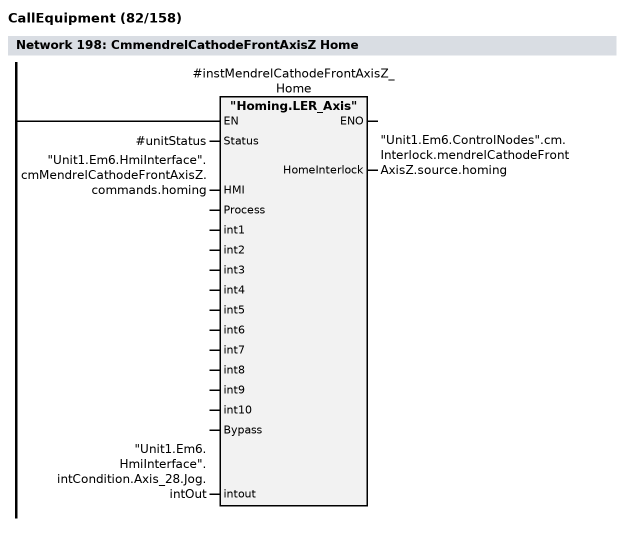
   RUNG wire#powerrail
      #instMendrelCathodeFrontAxisZ_Home(Status := #unitStatus, HMI := "Unit1.Em6.HmiInterface".cmMendrelCathodeFrontAxisZ.commands.homing, Process :=, int1 :=, int2 :=, int3 :=, int4 :=, int5 :=, int6 :=, int7 :=, int8 :=, int9 :=, int10 :=, Bypass :=, intout := "Unit1.Em6.HmiInterface".intCondition.Axis_28.Jog.intOut, HomeInterlock => "Unit1.Em6.ControlNodes".cm.Interlock.mendrelCathodeFrontAxisZ.source.homing)
   END_RUNG
   // the same network as SCL:
   #instMendrelCathodeFrontAxisZ_Home(Status := #unitStatus,   // "Homing.LER_Axis"
                           HMI := "Unit1.Em6.HmiInterface".cmMendrelCathodeFrontAxisZ.commands.homing,
                           intout := "Unit1.Em6.HmiInterface".intCondition.Axis_28.Jog.intOut,
                           HomeInterlock => "Unit1.Em6.ControlNodes".cm.Interlock.mendrelCathodeFrontAxisZ.source.homing);
END_REGION

REGION Network 199: CmmendrelCathodeFrontAxisZ Position Absolute Jog
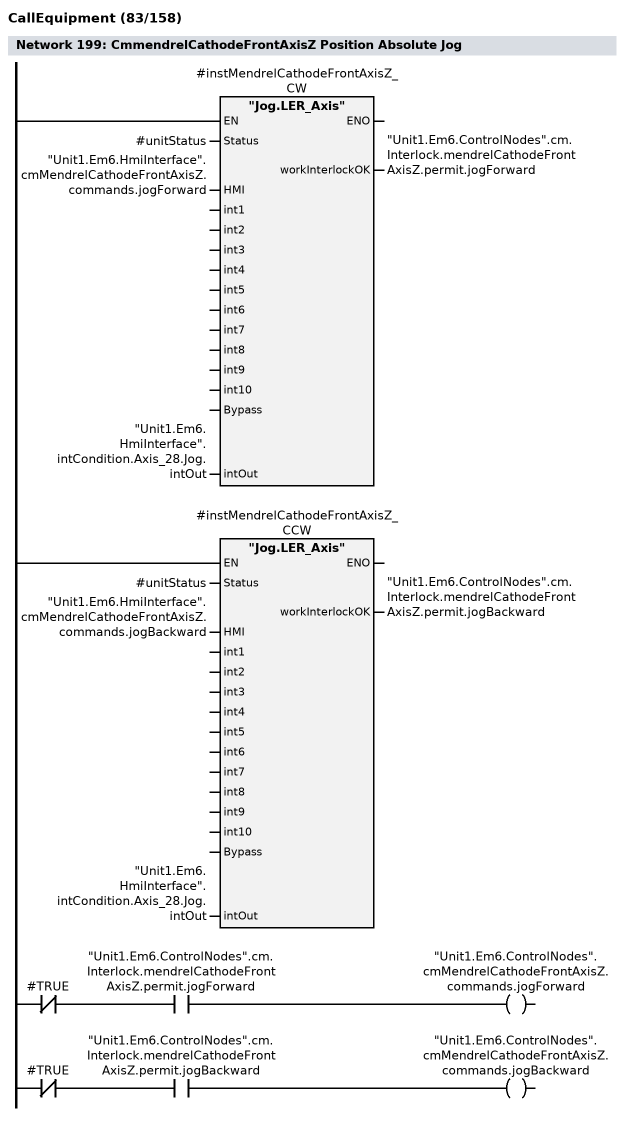
   RUNG wire#powerrail
      #instMendrelCathodeFrontAxisZ_CW(Status := #unitStatus, HMI := "Unit1.Em6.HmiInterface".cmMendrelCathodeFrontAxisZ.commands.jogForward, int1 :=, int2 :=, int3 :=, int4 :=, int5 :=, int6 :=, int7 :=, int8 :=, int9 :=, int10 :=, Bypass :=, intOut := "Unit1.Em6.HmiInterface".intCondition.Axis_28.Jog.intOut, workInterlockOK => "Unit1.Em6.ControlNodes".cm.Interlock.mendrelCathodeFrontAxisZ.permit.jogForward)
   END_RUNG
   RUNG wire#powerrail
      #instMendrelCathodeFrontAxisZ_CCW(Status := #unitStatus, HMI := "Unit1.Em6.HmiInterface".cmMendrelCathodeFrontAxisZ.commands.jogBackward, int1 :=, int2 :=, int3 :=, int4 :=, int5 :=, int6 :=, int7 :=, int8 :=, int9 :=, int10 :=, Bypass :=, intOut := "Unit1.Em6.HmiInterface".intCondition.Axis_28.Jog.intOut, workInterlockOK => "Unit1.Em6.ControlNodes".cm.Interlock.mendrelCathodeFrontAxisZ.permit.jogBackward)
   END_RUNG
   RUNG wire#powerrail
      I_Contact( #TRUE )
      Contact( "Unit1.Em6.ControlNodes".cm.Interlock.mendrelCathodeFrontAxisZ.permit.jogForward )
      Coil( "Unit1.Em6.ControlNodes".cmMendrelCathodeFrontAxisZ.commands.jogForward )
   END_RUNG
   RUNG wire#powerrail
      I_Contact( #TRUE )
      Contact( "Unit1.Em6.ControlNodes".cm.Interlock.mendrelCathodeFrontAxisZ.permit.jogBackward )
      Coil( "Unit1.Em6.ControlNodes".cmMendrelCathodeFrontAxisZ.commands.jogBackward )
   END_RUNG
   // the same network as SCL:
   #instMendrelCathodeFrontAxisZ_CW(Status := #unitStatus,   // "Jog.LER_Axis"
                           HMI := "Unit1.Em6.HmiInterface".cmMendrelCathodeFrontAxisZ.commands.jogForward,
                           intOut := "Unit1.Em6.HmiInterface".intCondition.Axis_28.Jog.intOut,
                           workInterlockOK => "Unit1.Em6.ControlNodes".cm.Interlock.mendrelCathodeFrontAxisZ.permit.jogForward);
   #instMendrelCathodeFrontAxisZ_CCW(Status := #unitStatus,   // "Jog.LER_Axis"
                           HMI := "Unit1.Em6.HmiInterface".cmMendrelCathodeFrontAxisZ.commands.jogBackward,
                           intOut := "Unit1.Em6.HmiInterface".intCondition.Axis_28.Jog.intOut,
                           workInterlockOK => "Unit1.Em6.ControlNodes".cm.Interlock.mendrelCathodeFrontAxisZ.permit.jogBackward);
   "Unit1.Em6.ControlNodes".cmMendrelCathodeFrontAxisZ.commands.jogForward := NOT #TRUE AND "Unit1.Em6.ControlNodes".cm.Interlock.mendrelCathodeFrontAxisZ.permit.jogForward;
   "Unit1.Em6.ControlNodes".cmMendrelCathodeFrontAxisZ.commands.jogBackward := NOT #TRUE AND "Unit1.Em6.ControlNodes".cm.Interlock.mendrelCathodeFrontAxisZ.permit.jogBackward;
END_REGION

REGION Network 200: CmmendrelCathodeFrontAxisZ Position Absolute Position0
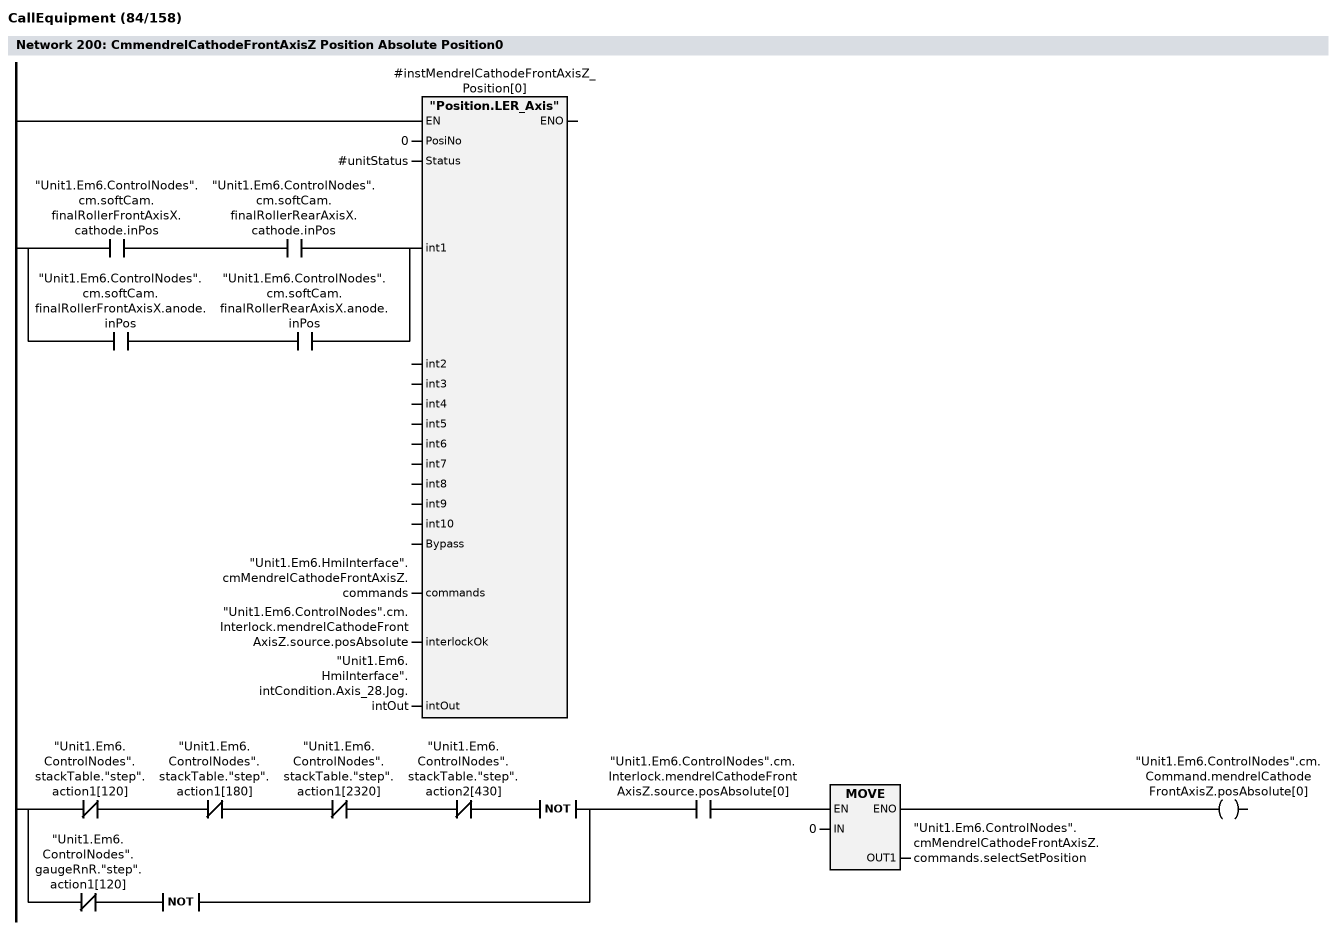
   RUNG wire#powerrail
      #instMendrelCathodeFrontAxisZ_Position[0](int1 := wire#w1, PosiNo := 0, Status := #unitStatus, int2 :=, int3 :=, int4 :=, int5 :=, int6 :=, int7 :=, int8 :=, int9 :=, int10 :=, Bypass :=, commands := "Unit1.Em6.HmiInterface".cmMendrelCathodeFrontAxisZ.commands, interlockOk := "Unit1.Em6.ControlNodes".cm.Interlock.mendrelCathodeFrontAxisZ.source.posAbsolute, intOut := "Unit1.Em6.HmiInterface".intCondition.Axis_28.Jog.intOut)
   END_RUNG
   RUNG wire#powerrail
      Contact( "Unit1.Em6.ControlNodes".cm.softCam.finalRollerFrontAxisX.cathode.inPos )
      Contact( "Unit1.Em6.ControlNodes".cm.softCam.finalRollerRearAxisX.cathode.inPos )
   END_RUNG wire#w1
   RUNG wire#powerrail
      Contact( "Unit1.Em6.ControlNodes".cm.softCam.finalRollerFrontAxisX.anode.inPos )
      Contact( "Unit1.Em6.ControlNodes".cm.softCam.finalRollerRearAxisX.anode.inPos )
   END_RUNG wire#w1
   RUNG wire#powerrail
      I_Contact( "Unit1.Em6.ControlNodes".stackTable."step".action1[120] )
      I_Contact( "Unit1.Em6.ControlNodes".stackTable."step".action1[180] )
      I_Contact( "Unit1.Em6.ControlNodes".stackTable."step".action1[2320] )
      I_Contact( "Unit1.Em6.ControlNodes".stackTable."step".action2[430] )
      Not()
      wire#w2
      Contact( "Unit1.Em6.ControlNodes".cm.Interlock.mendrelCathodeFrontAxisZ.source.posAbsolute[0] )
      Move(in := 0, out1 => "Unit1.Em6.ControlNodes".cmMendrelCathodeFrontAxisZ.commands.selectSetPosition)
      Coil( "Unit1.Em6.ControlNodes".cm.Command.mendrelCathodeFrontAxisZ.posAbsolute[0] )
   END_RUNG
   RUNG wire#powerrail
      I_Contact( "Unit1.Em6.ControlNodes".gaugeRnR."step".action1[120] )
      Not()
   END_RUNG wire#w2
   // the same network as SCL:
   #instMendrelCathodeFrontAxisZ_Position[0](PosiNo := 0,   // "Position.LER_Axis"
                           Status := #unitStatus,
                           int1 := ("Unit1.Em6.ControlNodes".cm.softCam.finalRollerFrontAxisX.cathode.inPos AND "Unit1.Em6.ControlNodes".cm.softCam.finalRollerRearAxisX.cathode.inPos) OR ("Unit1.Em6.ControlNodes".cm.softCam.finalRollerFrontAxisX.anode.inPos AND "Unit1.Em6.ControlNodes".cm.softCam.finalRollerRearAxisX.anode.inPos),
                           commands := "Unit1.Em6.HmiInterface".cmMendrelCathodeFrontAxisZ.commands,
                           interlockOk := "Unit1.Em6.ControlNodes".cm.Interlock.mendrelCathodeFrontAxisZ.source.posAbsolute,
                           intOut := "Unit1.Em6.HmiInterface".intCondition.Axis_28.Jog.intOut);
   #_w1 := (NOT (NOT "Unit1.Em6.ControlNodes".stackTable."step".action1[120] AND NOT "Unit1.Em6.ControlNodes".stackTable."step".action1[180] AND NOT "Unit1.Em6.ControlNodes".stackTable."step".action1[2320] AND NOT "Unit1.Em6.ControlNodes".stackTable."step".action2[430]) OR NOT (NOT "Unit1.Em6.ControlNodes".gaugeRnR."step".action1[120])) AND "Unit1.Em6.ControlNodes".cm.Interlock.mendrelCathodeFrontAxisZ.source.posAbsolute[0];
   IF #_w1 THEN "Unit1.Em6.ControlNodes".cmMendrelCathodeFrontAxisZ.commands.selectSetPosition := 0; END_IF;
   "Unit1.Em6.ControlNodes".cm.Command.mendrelCathodeFrontAxisZ.posAbsolute[0] := #_w1;
END_REGION

REGION Network 201: CmmendrelCathodeFrontAxisZ Position Absolute Position1
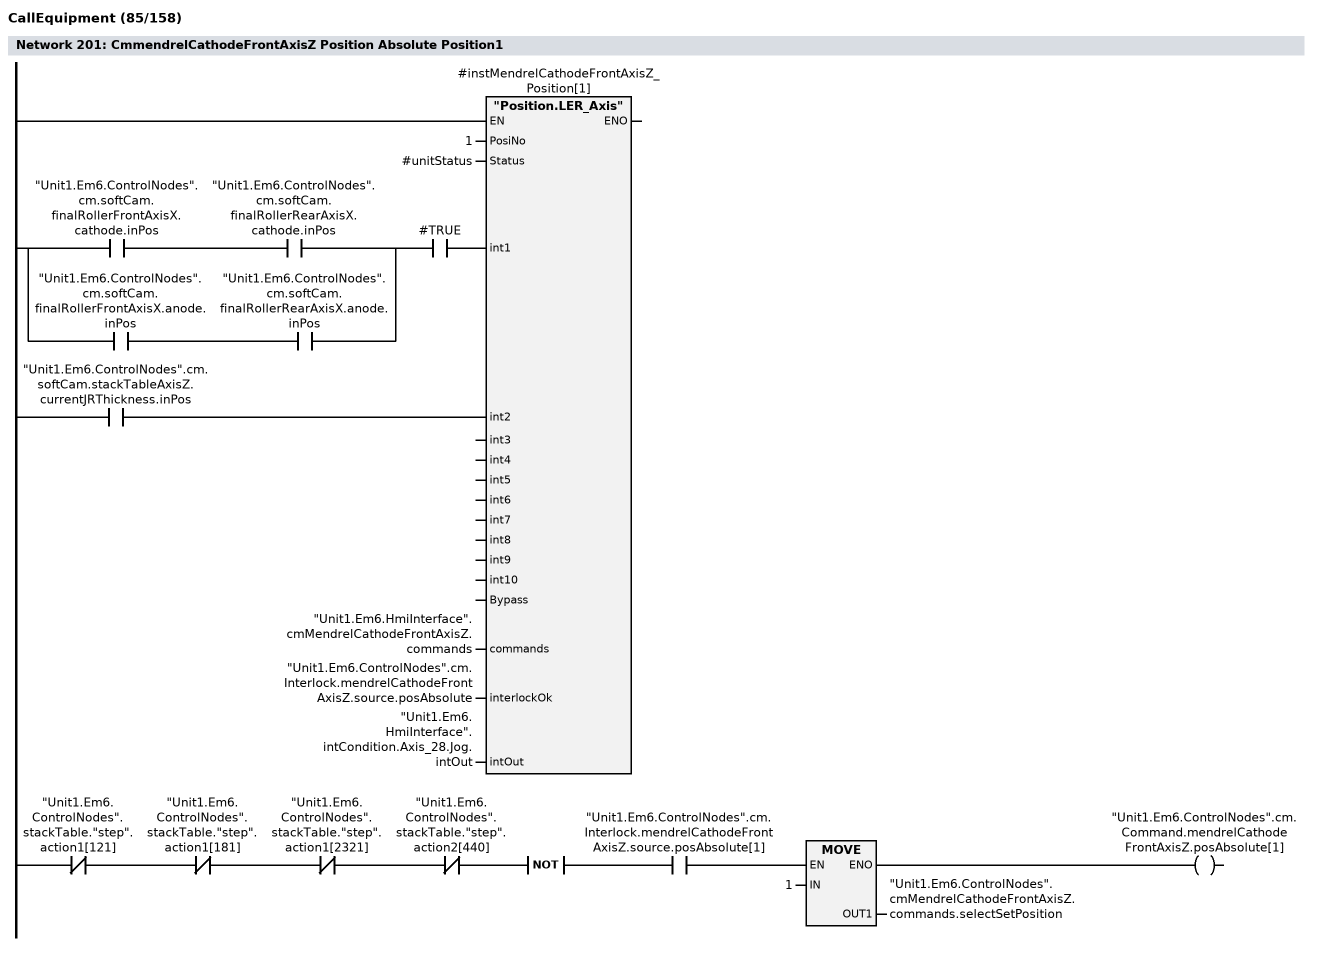
   RUNG wire#powerrail
      #instMendrelCathodeFrontAxisZ_Position[1](int1 := wire#w2, int2 := wire#w3, PosiNo := 1, Status := #unitStatus, int3 :=, int4 :=, int5 :=, int6 :=, int7 :=, int8 :=, int9 :=, int10 :=, Bypass :=, commands := "Unit1.Em6.HmiInterface".cmMendrelCathodeFrontAxisZ.commands, interlockOk := "Unit1.Em6.ControlNodes".cm.Interlock.mendrelCathodeFrontAxisZ.source.posAbsolute, intOut := "Unit1.Em6.HmiInterface".intCondition.Axis_28.Jog.intOut)
   END_RUNG
   RUNG wire#powerrail
      Contact( "Unit1.Em6.ControlNodes".cm.softCam.finalRollerFrontAxisX.cathode.inPos )
      Contact( "Unit1.Em6.ControlNodes".cm.softCam.finalRollerRearAxisX.cathode.inPos )
      wire#w1
      Contact( #TRUE )
   END_RUNG wire#w2
   RUNG wire#powerrail
      Contact( "Unit1.Em6.ControlNodes".cm.softCam.finalRollerFrontAxisX.anode.inPos )
      Contact( "Unit1.Em6.ControlNodes".cm.softCam.finalRollerRearAxisX.anode.inPos )
   END_RUNG wire#w1
   RUNG wire#powerrail
      Contact( "Unit1.Em6.ControlNodes".cm.softCam.stackTableAxisZ.currentJRThickness.inPos )
   END_RUNG wire#w3
   RUNG wire#powerrail
      I_Contact( "Unit1.Em6.ControlNodes".stackTable."step".action1[121] )
      I_Contact( "Unit1.Em6.ControlNodes".stackTable."step".action1[181] )
      I_Contact( "Unit1.Em6.ControlNodes".stackTable."step".action1[2321] )
      I_Contact( "Unit1.Em6.ControlNodes".stackTable."step".action2[440] )
      Not()
      Contact( "Unit1.Em6.ControlNodes".cm.Interlock.mendrelCathodeFrontAxisZ.source.posAbsolute[1] )
      Move(in := 1, out1 => "Unit1.Em6.ControlNodes".cmMendrelCathodeFrontAxisZ.commands.selectSetPosition)
      Coil( "Unit1.Em6.ControlNodes".cm.Command.mendrelCathodeFrontAxisZ.posAbsolute[1] )
   END_RUNG
   // the same network as SCL:
   #instMendrelCathodeFrontAxisZ_Position[1](PosiNo := 1,   // "Position.LER_Axis"
                           Status := #unitStatus,
                           int1 := (("Unit1.Em6.ControlNodes".cm.softCam.finalRollerFrontAxisX.cathode.inPos AND "Unit1.Em6.ControlNodes".cm.softCam.finalRollerRearAxisX.cathode.inPos) OR ("Unit1.Em6.ControlNodes".cm.softCam.finalRollerFrontAxisX.anode.inPos AND "Unit1.Em6.ControlNodes".cm.softCam.finalRollerRearAxisX.anode.inPos)) AND #TRUE,
                           int2 := "Unit1.Em6.ControlNodes".cm.softCam.stackTableAxisZ.currentJRThickness.inPos,
                           commands := "Unit1.Em6.HmiInterface".cmMendrelCathodeFrontAxisZ.commands,
                           interlockOk := "Unit1.Em6.ControlNodes".cm.Interlock.mendrelCathodeFrontAxisZ.source.posAbsolute,
                           intOut := "Unit1.Em6.HmiInterface".intCondition.Axis_28.Jog.intOut);
   #_w1 := NOT (NOT "Unit1.Em6.ControlNodes".stackTable."step".action1[121] AND NOT "Unit1.Em6.ControlNodes".stackTable."step".action1[181] AND NOT "Unit1.Em6.ControlNodes".stackTable."step".action1[2321] AND NOT "Unit1.Em6.ControlNodes".stackTable."step".action2[440]) AND "Unit1.Em6.ControlNodes".cm.Interlock.mendrelCathodeFrontAxisZ.source.posAbsolute[1];
   IF #_w1 THEN "Unit1.Em6.ControlNodes".cmMendrelCathodeFrontAxisZ.commands.selectSetPosition := 1; END_IF;
   "Unit1.Em6.ControlNodes".cm.Command.mendrelCathodeFrontAxisZ.posAbsolute[1] := #_w1;
END_REGION

REGION Network 202: CmmendrelCathodeFrontAxisZ Position Absolute Position2
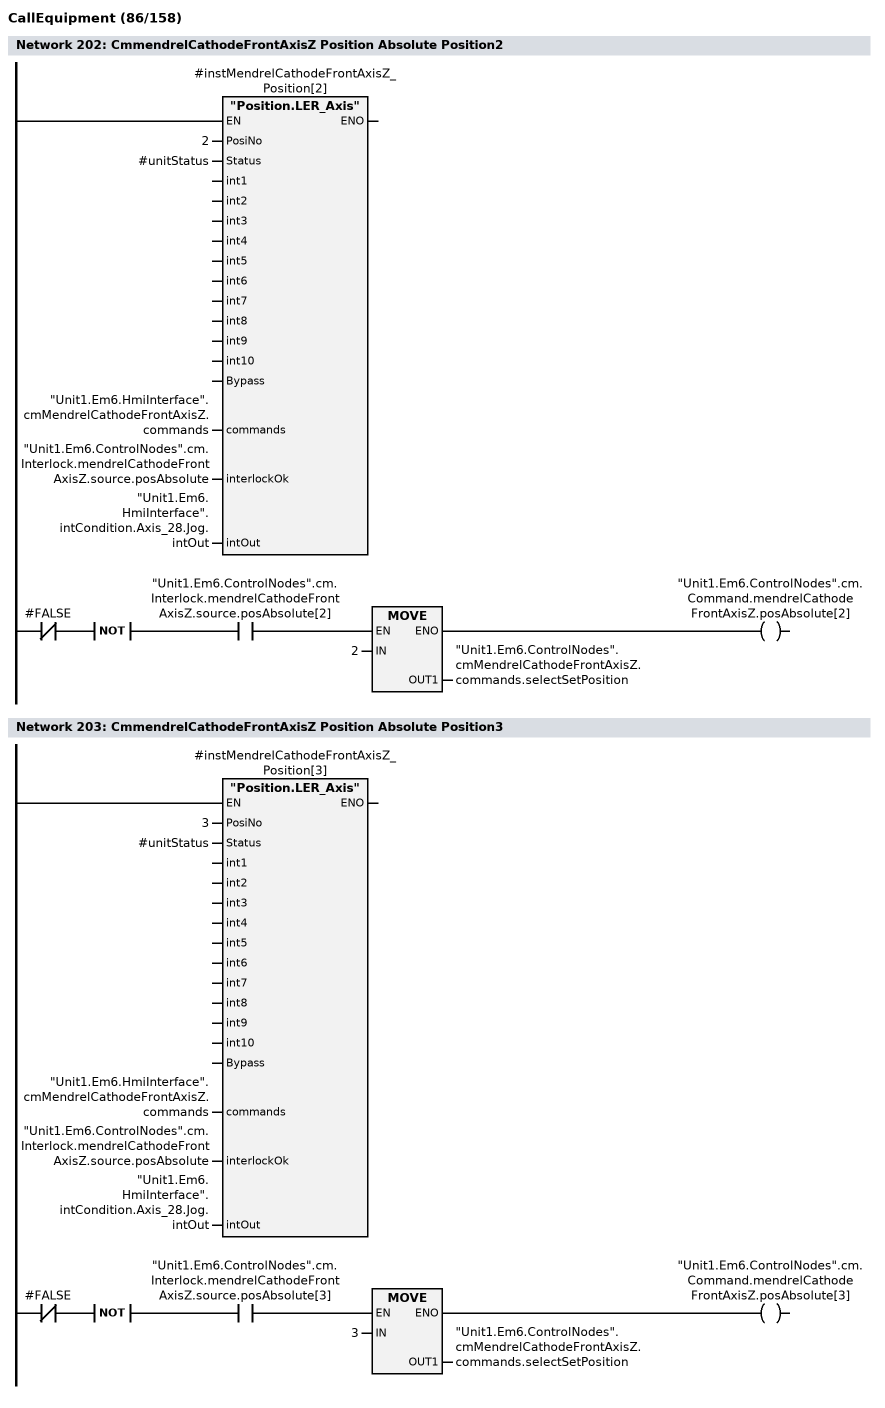
   RUNG wire#powerrail
      #instMendrelCathodeFrontAxisZ_Position[2](PosiNo := 2, Status := #unitStatus, int1 :=, int2 :=, int3 :=, int4 :=, int5 :=, int6 :=, int7 :=, int8 :=, int9 :=, int10 :=, Bypass :=, commands := "Unit1.Em6.HmiInterface".cmMendrelCathodeFrontAxisZ.commands, interlockOk := "Unit1.Em6.ControlNodes".cm.Interlock.mendrelCathodeFrontAxisZ.source.posAbsolute, intOut := "Unit1.Em6.HmiInterface".intCondition.Axis_28.Jog.intOut)
   END_RUNG
   RUNG wire#powerrail
      I_Contact( #FALSE )
      Not()
      Contact( "Unit1.Em6.ControlNodes".cm.Interlock.mendrelCathodeFrontAxisZ.source.posAbsolute[2] )
      Move(in := 2, out1 => "Unit1.Em6.ControlNodes".cmMendrelCathodeFrontAxisZ.commands.selectSetPosition)
      Coil( "Unit1.Em6.ControlNodes".cm.Command.mendrelCathodeFrontAxisZ.posAbsolute[2] )
   END_RUNG
   // the same network as SCL:
   #instMendrelCathodeFrontAxisZ_Position[2](PosiNo := 2,   // "Position.LER_Axis"
                           Status := #unitStatus,
                           commands := "Unit1.Em6.HmiInterface".cmMendrelCathodeFrontAxisZ.commands,
                           interlockOk := "Unit1.Em6.ControlNodes".cm.Interlock.mendrelCathodeFrontAxisZ.source.posAbsolute,
                           intOut := "Unit1.Em6.HmiInterface".intCondition.Axis_28.Jog.intOut);
   #_w1 := NOT (NOT #FALSE) AND "Unit1.Em6.ControlNodes".cm.Interlock.mendrelCathodeFrontAxisZ.source.posAbsolute[2];
   IF #_w1 THEN "Unit1.Em6.ControlNodes".cmMendrelCathodeFrontAxisZ.commands.selectSetPosition := 2; END_IF;
   "Unit1.Em6.ControlNodes".cm.Command.mendrelCathodeFrontAxisZ.posAbsolute[2] := #_w1;
END_REGION

REGION Network 203: CmmendrelCathodeFrontAxisZ Position Absolute Position3
   RUNG wire#powerrail
      #instMendrelCathodeFrontAxisZ_Position[3](PosiNo := 3, Status := #unitStatus, int1 :=, int2 :=, int3 :=, int4 :=, int5 :=, int6 :=, int7 :=, int8 :=, int9 :=, int10 :=, Bypass :=, commands := "Unit1.Em6.HmiInterface".cmMendrelCathodeFrontAxisZ.commands, interlockOk := "Unit1.Em6.ControlNodes".cm.Interlock.mendrelCathodeFrontAxisZ.source.posAbsolute, intOut := "Unit1.Em6.HmiInterface".intCondition.Axis_28.Jog.intOut)
   END_RUNG
   RUNG wire#powerrail
      I_Contact( #FALSE )
      Not()
      Contact( "Unit1.Em6.ControlNodes".cm.Interlock.mendrelCathodeFrontAxisZ.source.posAbsolute[3] )
      Move(in := 3, out1 => "Unit1.Em6.ControlNodes".cmMendrelCathodeFrontAxisZ.commands.selectSetPosition)
      Coil( "Unit1.Em6.ControlNodes".cm.Command.mendrelCathodeFrontAxisZ.posAbsolute[3] )
   END_RUNG
   // the same network as SCL:
   #instMendrelCathodeFrontAxisZ_Position[3](PosiNo := 3,   // "Position.LER_Axis"
                           Status := #unitStatus,
                           commands := "Unit1.Em6.HmiInterface".cmMendrelCathodeFrontAxisZ.commands,
                           interlockOk := "Unit1.Em6.ControlNodes".cm.Interlock.mendrelCathodeFrontAxisZ.source.posAbsolute,
                           intOut := "Unit1.Em6.HmiInterface".intCondition.Axis_28.Jog.intOut);
   #_w1 := NOT (NOT #FALSE) AND "Unit1.Em6.ControlNodes".cm.Interlock.mendrelCathodeFrontAxisZ.source.posAbsolute[3];
   IF #_w1 THEN "Unit1.Em6.ControlNodes".cmMendrelCathodeFrontAxisZ.commands.selectSetPosition := 3; END_IF;
   "Unit1.Em6.ControlNodes".cm.Command.mendrelCathodeFrontAxisZ.posAbsolute[3] := #_w1;
END_REGION

REGION Network 204: CmmendrelCathodeFrontAxisZ Position Absolute Position4
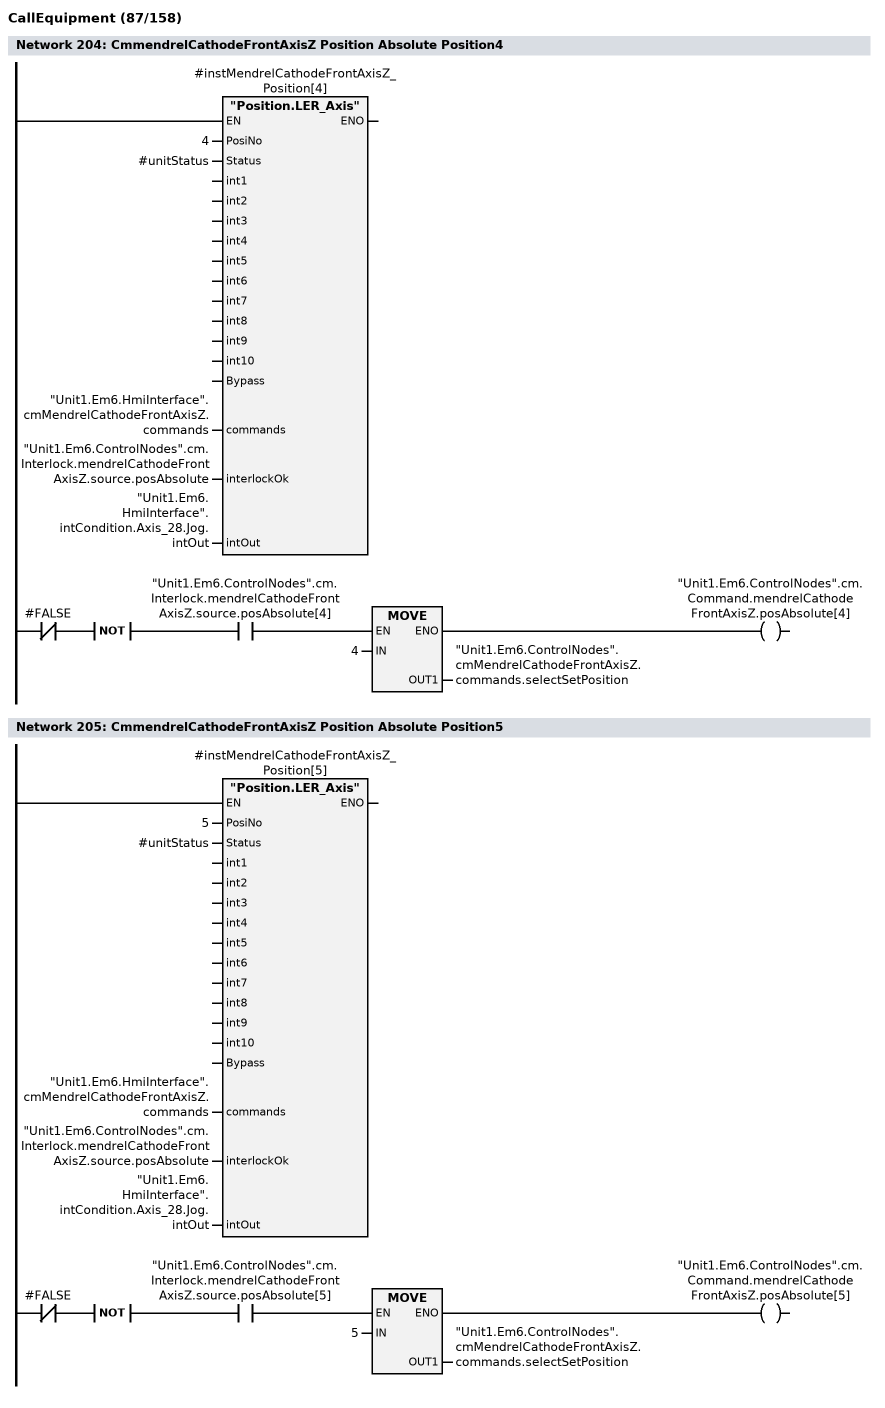
   RUNG wire#powerrail
      #instMendrelCathodeFrontAxisZ_Position[4](PosiNo := 4, Status := #unitStatus, int1 :=, int2 :=, int3 :=, int4 :=, int5 :=, int6 :=, int7 :=, int8 :=, int9 :=, int10 :=, Bypass :=, commands := "Unit1.Em6.HmiInterface".cmMendrelCathodeFrontAxisZ.commands, interlockOk := "Unit1.Em6.ControlNodes".cm.Interlock.mendrelCathodeFrontAxisZ.source.posAbsolute, intOut := "Unit1.Em6.HmiInterface".intCondition.Axis_28.Jog.intOut)
   END_RUNG
   RUNG wire#powerrail
      I_Contact( #FALSE )
      Not()
      Contact( "Unit1.Em6.ControlNodes".cm.Interlock.mendrelCathodeFrontAxisZ.source.posAbsolute[4] )
      Move(in := 4, out1 => "Unit1.Em6.ControlNodes".cmMendrelCathodeFrontAxisZ.commands.selectSetPosition)
      Coil( "Unit1.Em6.ControlNodes".cm.Command.mendrelCathodeFrontAxisZ.posAbsolute[4] )
   END_RUNG
   // the same network as SCL:
   #instMendrelCathodeFrontAxisZ_Position[4](PosiNo := 4,   // "Position.LER_Axis"
                           Status := #unitStatus,
                           commands := "Unit1.Em6.HmiInterface".cmMendrelCathodeFrontAxisZ.commands,
                           interlockOk := "Unit1.Em6.ControlNodes".cm.Interlock.mendrelCathodeFrontAxisZ.source.posAbsolute,
                           intOut := "Unit1.Em6.HmiInterface".intCondition.Axis_28.Jog.intOut);
   #_w1 := NOT (NOT #FALSE) AND "Unit1.Em6.ControlNodes".cm.Interlock.mendrelCathodeFrontAxisZ.source.posAbsolute[4];
   IF #_w1 THEN "Unit1.Em6.ControlNodes".cmMendrelCathodeFrontAxisZ.commands.selectSetPosition := 4; END_IF;
   "Unit1.Em6.ControlNodes".cm.Command.mendrelCathodeFrontAxisZ.posAbsolute[4] := #_w1;
END_REGION

REGION Network 205: CmmendrelCathodeFrontAxisZ Position Absolute Position5
   RUNG wire#powerrail
      #instMendrelCathodeFrontAxisZ_Position[5](PosiNo := 5, Status := #unitStatus, int1 :=, int2 :=, int3 :=, int4 :=, int5 :=, int6 :=, int7 :=, int8 :=, int9 :=, int10 :=, Bypass :=, commands := "Unit1.Em6.HmiInterface".cmMendrelCathodeFrontAxisZ.commands, interlockOk := "Unit1.Em6.ControlNodes".cm.Interlock.mendrelCathodeFrontAxisZ.source.posAbsolute, intOut := "Unit1.Em6.HmiInterface".intCondition.Axis_28.Jog.intOut)
   END_RUNG
   RUNG wire#powerrail
      I_Contact( #FALSE )
      Not()
      Contact( "Unit1.Em6.ControlNodes".cm.Interlock.mendrelCathodeFrontAxisZ.source.posAbsolute[5] )
      Move(in := 5, out1 => "Unit1.Em6.ControlNodes".cmMendrelCathodeFrontAxisZ.commands.selectSetPosition)
      Coil( "Unit1.Em6.ControlNodes".cm.Command.mendrelCathodeFrontAxisZ.posAbsolute[5] )
   END_RUNG
   // the same network as SCL:
   #instMendrelCathodeFrontAxisZ_Position[5](PosiNo := 5,   // "Position.LER_Axis"
                           Status := #unitStatus,
                           commands := "Unit1.Em6.HmiInterface".cmMendrelCathodeFrontAxisZ.commands,
                           interlockOk := "Unit1.Em6.ControlNodes".cm.Interlock.mendrelCathodeFrontAxisZ.source.posAbsolute,
                           intOut := "Unit1.Em6.HmiInterface".intCondition.Axis_28.Jog.intOut);
   #_w1 := NOT (NOT #FALSE) AND "Unit1.Em6.ControlNodes".cm.Interlock.mendrelCathodeFrontAxisZ.source.posAbsolute[5];
   IF #_w1 THEN "Unit1.Em6.ControlNodes".cmMendrelCathodeFrontAxisZ.commands.selectSetPosition := 5; END_IF;
   "Unit1.Em6.ControlNodes".cm.Command.mendrelCathodeFrontAxisZ.posAbsolute[5] := #_w1;
END_REGION

REGION Network 206: CmmendrelCathodeFrontAxisZ Summary Command
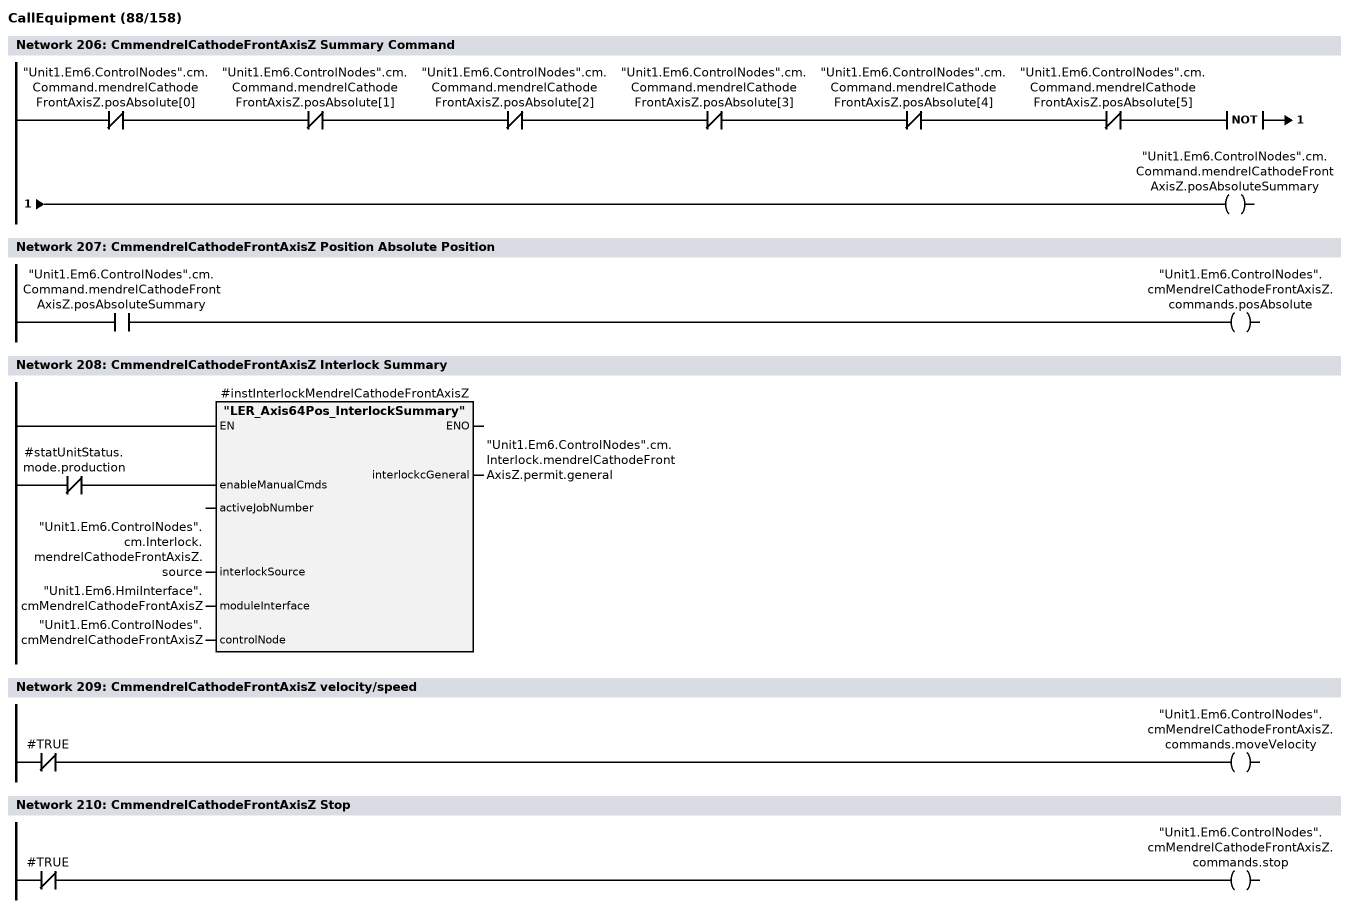
   RUNG wire#powerrail
      I_Contact( "Unit1.Em6.ControlNodes".cm.Command.mendrelCathodeFrontAxisZ.posAbsolute[0] )
      I_Contact( "Unit1.Em6.ControlNodes".cm.Command.mendrelCathodeFrontAxisZ.posAbsolute[1] )
      I_Contact( "Unit1.Em6.ControlNodes".cm.Command.mendrelCathodeFrontAxisZ.posAbsolute[2] )
      I_Contact( "Unit1.Em6.ControlNodes".cm.Command.mendrelCathodeFrontAxisZ.posAbsolute[3] )
      I_Contact( "Unit1.Em6.ControlNodes".cm.Command.mendrelCathodeFrontAxisZ.posAbsolute[4] )
      I_Contact( "Unit1.Em6.ControlNodes".cm.Command.mendrelCathodeFrontAxisZ.posAbsolute[5] )
      Not()
      Coil( "Unit1.Em6.ControlNodes".cm.Command.mendrelCathodeFrontAxisZ.posAbsoluteSummary )
   END_RUNG
   // the same network as SCL:
   "Unit1.Em6.ControlNodes".cm.Command.mendrelCathodeFrontAxisZ.posAbsoluteSummary := NOT (NOT "Unit1.Em6.ControlNodes".cm.Command.mendrelCathodeFrontAxisZ.posAbsolute[0] AND NOT "Unit1.Em6.ControlNodes".cm.Command.mendrelCathodeFrontAxisZ.posAbsolute[1] AND NOT "Unit1.Em6.ControlNodes".cm.Command.mendrelCathodeFrontAxisZ.posAbsolute[2] AND NOT "Unit1.Em6.ControlNodes".cm.Command.mendrelCathodeFrontAxisZ.posAbsolute[3] AND NOT "Unit1.Em6.ControlNodes".cm.Command.mendrelCathodeFrontAxisZ.posAbsolute[4] AND NOT "Unit1.Em6.ControlNodes".cm.Command.mendrelCathodeFrontAxisZ.posAbsolute[5]);
END_REGION

REGION Network 207: CmmendrelCathodeFrontAxisZ Position Absolute Position
   RUNG wire#powerrail
      Contact( "Unit1.Em6.ControlNodes".cm.Command.mendrelCathodeFrontAxisZ.posAbsoluteSummary )
      Coil( "Unit1.Em6.ControlNodes".cmMendrelCathodeFrontAxisZ.commands.posAbsolute )
   END_RUNG
   // the same network as SCL:
   "Unit1.Em6.ControlNodes".cmMendrelCathodeFrontAxisZ.commands.posAbsolute := "Unit1.Em6.ControlNodes".cm.Command.mendrelCathodeFrontAxisZ.posAbsoluteSummary;
END_REGION

REGION Network 208: CmmendrelCathodeFrontAxisZ Interlock Summary
   RUNG wire#powerrail
      #instInterlockMendrelCathodeFrontAxisZ(enableManualCmds := wire#w1, activeJobNumber :=, interlockSource := "Unit1.Em6.ControlNodes".cm.Interlock.mendrelCathodeFrontAxisZ.source, moduleInterface := "Unit1.Em6.HmiInterface".cmMendrelCathodeFrontAxisZ, controlNode := "Unit1.Em6.ControlNodes".cmMendrelCathodeFrontAxisZ, interlockcGeneral => "Unit1.Em6.ControlNodes".cm.Interlock.mendrelCathodeFrontAxisZ.permit.general)
   END_RUNG
   RUNG wire#powerrail
      I_Contact( #statUnitStatus.mode.production )
   END_RUNG wire#w1
   // the same network as SCL:
   #instInterlockMendrelCathodeFrontAxisZ(enableManualCmds := NOT #statUnitStatus.mode.production,   // "LER_Axis64Pos_InterlockSummary"
                           interlockSource := "Unit1.Em6.ControlNodes".cm.Interlock.mendrelCathodeFrontAxisZ.source,
                           moduleInterface := "Unit1.Em6.HmiInterface".cmMendrelCathodeFrontAxisZ,
                           controlNode := "Unit1.Em6.ControlNodes".cmMendrelCathodeFrontAxisZ,
                           interlockcGeneral => "Unit1.Em6.ControlNodes".cm.Interlock.mendrelCathodeFrontAxisZ.permit.general);
END_REGION

REGION Network 209: CmmendrelCathodeFrontAxisZ velocity/speed
   RUNG wire#powerrail
      I_Contact( #TRUE )
      Coil( "Unit1.Em6.ControlNodes".cmMendrelCathodeFrontAxisZ.commands.moveVelocity )
   END_RUNG
   // the same network as SCL:
   "Unit1.Em6.ControlNodes".cmMendrelCathodeFrontAxisZ.commands.moveVelocity := NOT #TRUE;
END_REGION

REGION Network 210: CmmendrelCathodeFrontAxisZ Stop
   RUNG wire#powerrail
      I_Contact( #TRUE )
      Coil( "Unit1.Em6.ControlNodes".cmMendrelCathodeFrontAxisZ.commands.stop )
   END_RUNG
   // the same network as SCL:
   "Unit1.Em6.ControlNodes".cmMendrelCathodeFrontAxisZ.commands.stop := NOT #TRUE;
END_REGION

REGION Network 211: Call CM Cathode Mandrel Front Z-Axis (LBC_Axis64Pos)
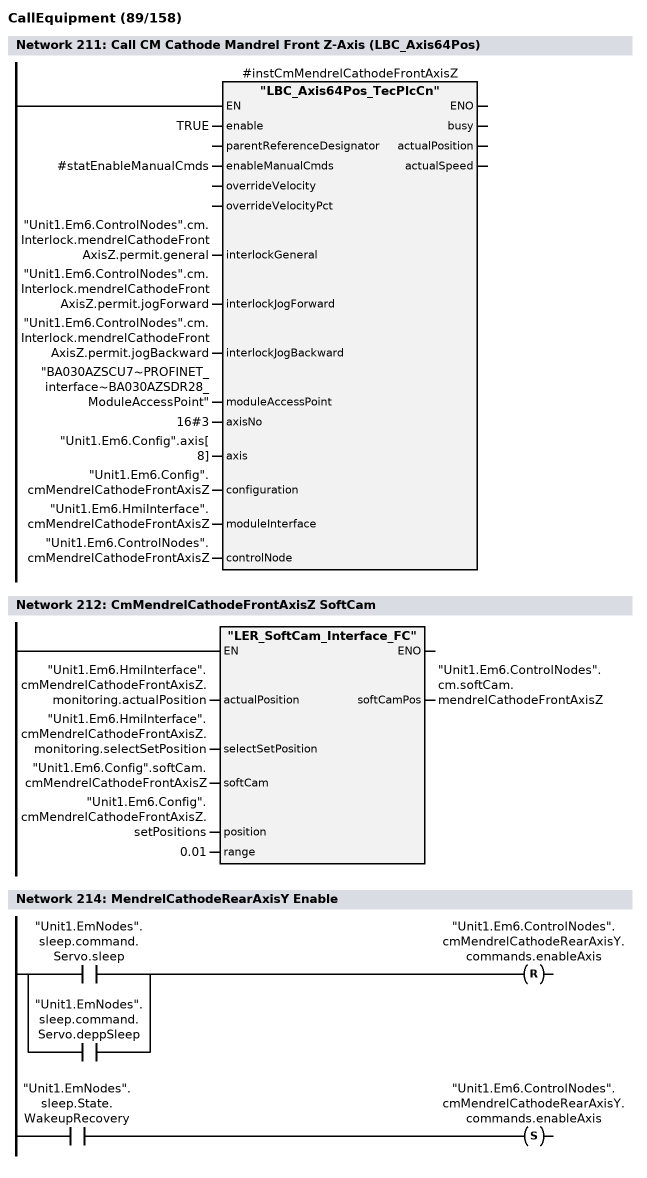
   RUNG wire#powerrail
      #instCmMendrelCathodeFrontAxisZ(enable := TRUE, parentReferenceDesignator :=, enableManualCmds := #statEnableManualCmds, overrideVelocity :=, overrideVelocityPct :=, interlockGeneral := "Unit1.Em6.ControlNodes".cm.Interlock.mendrelCathodeFrontAxisZ.permit.general, interlockJogForward := "Unit1.Em6.ControlNodes".cm.Interlock.mendrelCathodeFrontAxisZ.permit.jogForward, interlockJogBackward := "Unit1.Em6.ControlNodes".cm.Interlock.mendrelCathodeFrontAxisZ.permit.jogBackward, moduleAccessPoint := "BA030AZSCU7~PROFINET_interface~BA030AZSDR28_ModuleAccessPoint", axisNo := 16#3, axis := "Unit1.Em6.Config".axis[8], configuration := "Unit1.Em6.Config".cmMendrelCathodeFrontAxisZ, moduleInterface := "Unit1.Em6.HmiInterface".cmMendrelCathodeFrontAxisZ, controlNode := "Unit1.Em6.ControlNodes".cmMendrelCathodeFrontAxisZ, busy =>, actualPosition =>, actualSpeed =>)
   END_RUNG
   // the same network as SCL:
   #instCmMendrelCathodeFrontAxisZ(enable := TRUE,   // "LBC_Axis64Pos_TecPlcCn"
                           enableManualCmds := #statEnableManualCmds,
                           interlockGeneral := "Unit1.Em6.ControlNodes".cm.Interlock.mendrelCathodeFrontAxisZ.permit.general,
                           interlockJogForward := "Unit1.Em6.ControlNodes".cm.Interlock.mendrelCathodeFrontAxisZ.permit.jogForward,
                           interlockJogBackward := "Unit1.Em6.ControlNodes".cm.Interlock.mendrelCathodeFrontAxisZ.permit.jogBackward,
                           moduleAccessPoint := "BA030AZSCU7~PROFINET_interface~BA030AZSDR28_ModuleAccessPoint",
                           axisNo := 16#3,
                           axis := "Unit1.Em6.Config".axis[8],
                           configuration := "Unit1.Em6.Config".cmMendrelCathodeFrontAxisZ,
                           moduleInterface := "Unit1.Em6.HmiInterface".cmMendrelCathodeFrontAxisZ,
                           controlNode := "Unit1.Em6.ControlNodes".cmMendrelCathodeFrontAxisZ);
END_REGION

REGION Network 212: CmMendrelCathodeFrontAxisZ SoftCam
   RUNG wire#powerrail
      "LER_SoftCam_Interface_FC"(actualPosition := "Unit1.Em6.HmiInterface".cmMendrelCathodeFrontAxisZ.monitoring.actualPosition, selectSetPosition := "Unit1.Em6.HmiInterface".cmMendrelCathodeFrontAxisZ.monitoring.selectSetPosition, softCam := "Unit1.Em6.Config".softCam.cmMendrelCathodeFrontAxisZ, position := "Unit1.Em6.Config".cmMendrelCathodeFrontAxisZ.setPositions, range := 0.01, softCamPos => "Unit1.Em6.ControlNodes".cm.softCam.mendrelCathodeFrontAxisZ)
   END_RUNG
   // the same network as SCL:
   "LER_SoftCam_Interface_FC"(actualPosition := "Unit1.Em6.HmiInterface".cmMendrelCathodeFrontAxisZ.monitoring.actualPosition,
                           selectSetPosition := "Unit1.Em6.HmiInterface".cmMendrelCathodeFrontAxisZ.monitoring.selectSetPosition,
                           softCam := "Unit1.Em6.Config".softCam.cmMendrelCathodeFrontAxisZ,
                           position := "Unit1.Em6.Config".cmMendrelCathodeFrontAxisZ.setPositions,
                           range := 0.01,
                           softCamPos => "Unit1.Em6.ControlNodes".cm.softCam.mendrelCathodeFrontAxisZ);
END_REGION

REGION Network 214: MendrelCathodeRearAxisY Enable
   RUNG wire#powerrail
      Contact( "Unit1.EmNodes".sleep.command.Servo.sleep )
      wire#w1
      R_Coil( "Unit1.Em6.ControlNodes".cmMendrelCathodeRearAxisY.commands.enableAxis )
   END_RUNG
   RUNG wire#powerrail
      Contact( "Unit1.EmNodes".sleep.command.Servo.deppSleep )
   END_RUNG wire#w1
   RUNG wire#powerrail
      Contact( "Unit1.EmNodes".sleep.State.WakeupRecovery )
      S_Coil( "Unit1.Em6.ControlNodes".cmMendrelCathodeRearAxisY.commands.enableAxis )
   END_RUNG
   // the same network as SCL:
   IF "Unit1.EmNodes".sleep.command.Servo.sleep OR "Unit1.EmNodes".sleep.command.Servo.deppSleep THEN
       "Unit1.Em6.ControlNodes".cmMendrelCathodeRearAxisY.commands.enableAxis := FALSE;
   END_IF;
   IF "Unit1.EmNodes".sleep.State.WakeupRecovery THEN
       "Unit1.Em6.ControlNodes".cmMendrelCathodeRearAxisY.commands.enableAxis := TRUE;
   END_IF;
END_REGION

REGION Network 215: CmmendrelCathodeRearAxisY Home
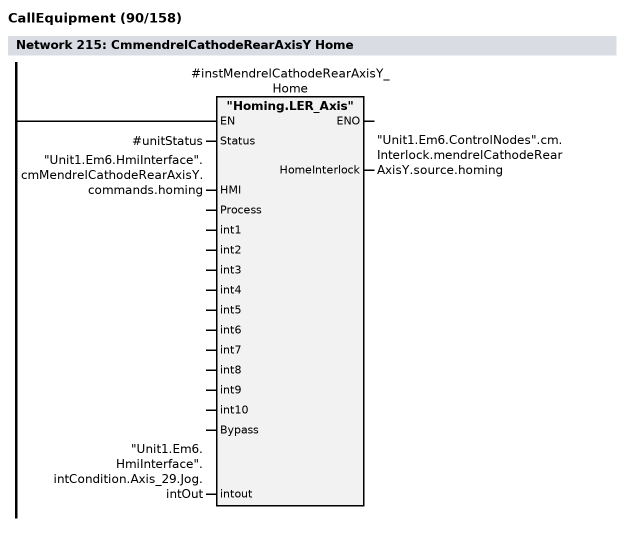
   RUNG wire#powerrail
      #instMendrelCathodeRearAxisY_Home(Status := #unitStatus, HMI := "Unit1.Em6.HmiInterface".cmMendrelCathodeRearAxisY.commands.homing, Process :=, int1 :=, int2 :=, int3 :=, int4 :=, int5 :=, int6 :=, int7 :=, int8 :=, int9 :=, int10 :=, Bypass :=, intout := "Unit1.Em6.HmiInterface".intCondition.Axis_29.Jog.intOut, HomeInterlock => "Unit1.Em6.ControlNodes".cm.Interlock.mendrelCathodeRearAxisY.source.homing)
   END_RUNG
   // the same network as SCL:
   #instMendrelCathodeRearAxisY_Home(Status := #unitStatus,   // "Homing.LER_Axis"
                           HMI := "Unit1.Em6.HmiInterface".cmMendrelCathodeRearAxisY.commands.homing,
                           intout := "Unit1.Em6.HmiInterface".intCondition.Axis_29.Jog.intOut,
                           HomeInterlock => "Unit1.Em6.ControlNodes".cm.Interlock.mendrelCathodeRearAxisY.source.homing);
END_REGION

REGION Network 216: CmMendrelCathodeRearAxisY Position Absolute Jog
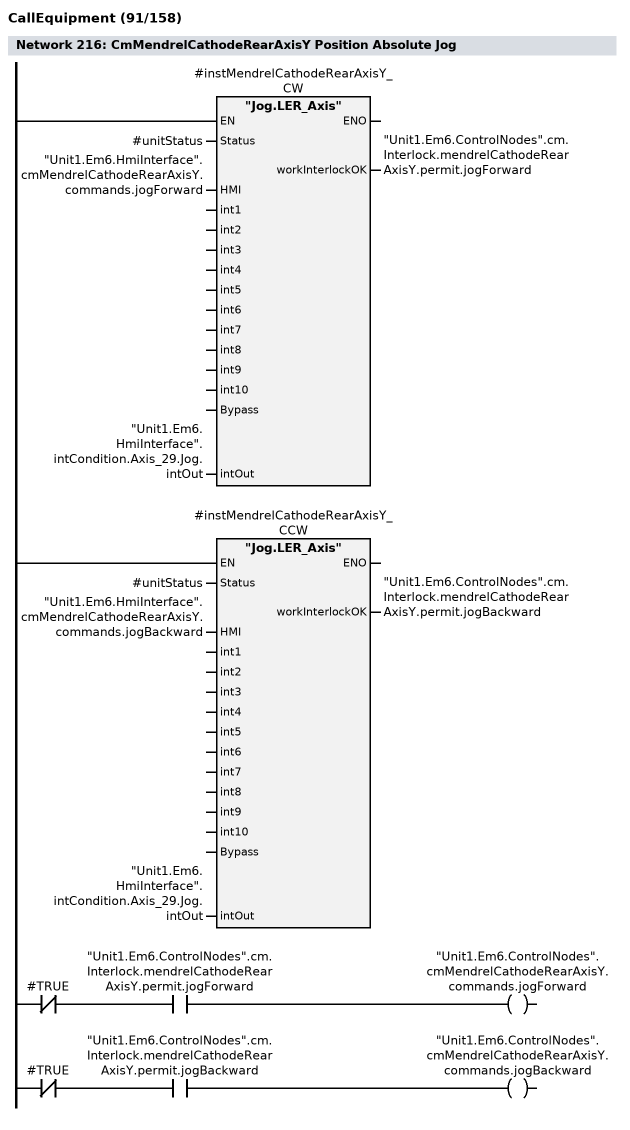
   RUNG wire#powerrail
      #instMendrelCathodeRearAxisY_CW(Status := #unitStatus, HMI := "Unit1.Em6.HmiInterface".cmMendrelCathodeRearAxisY.commands.jogForward, int1 :=, int2 :=, int3 :=, int4 :=, int5 :=, int6 :=, int7 :=, int8 :=, int9 :=, int10 :=, Bypass :=, intOut := "Unit1.Em6.HmiInterface".intCondition.Axis_29.Jog.intOut, workInterlockOK => "Unit1.Em6.ControlNodes".cm.Interlock.mendrelCathodeRearAxisY.permit.jogForward)
   END_RUNG
   RUNG wire#powerrail
      #instMendrelCathodeRearAxisY_CCW(Status := #unitStatus, HMI := "Unit1.Em6.HmiInterface".cmMendrelCathodeRearAxisY.commands.jogBackward, int1 :=, int2 :=, int3 :=, int4 :=, int5 :=, int6 :=, int7 :=, int8 :=, int9 :=, int10 :=, Bypass :=, intOut := "Unit1.Em6.HmiInterface".intCondition.Axis_29.Jog.intOut, workInterlockOK => "Unit1.Em6.ControlNodes".cm.Interlock.mendrelCathodeRearAxisY.permit.jogBackward)
   END_RUNG
   RUNG wire#powerrail
      I_Contact( #TRUE )
      Contact( "Unit1.Em6.ControlNodes".cm.Interlock.mendrelCathodeRearAxisY.permit.jogForward )
      Coil( "Unit1.Em6.ControlNodes".cmMendrelCathodeRearAxisY.commands.jogForward )
   END_RUNG
   RUNG wire#powerrail
      I_Contact( #TRUE )
      Contact( "Unit1.Em6.ControlNodes".cm.Interlock.mendrelCathodeRearAxisY.permit.jogBackward )
      Coil( "Unit1.Em6.ControlNodes".cmMendrelCathodeRearAxisY.commands.jogBackward )
   END_RUNG
   // the same network as SCL:
   #instMendrelCathodeRearAxisY_CW(Status := #unitStatus,   // "Jog.LER_Axis"
                           HMI := "Unit1.Em6.HmiInterface".cmMendrelCathodeRearAxisY.commands.jogForward,
                           intOut := "Unit1.Em6.HmiInterface".intCondition.Axis_29.Jog.intOut,
                           workInterlockOK => "Unit1.Em6.ControlNodes".cm.Interlock.mendrelCathodeRearAxisY.permit.jogForward);
   #instMendrelCathodeRearAxisY_CCW(Status := #unitStatus,   // "Jog.LER_Axis"
                           HMI := "Unit1.Em6.HmiInterface".cmMendrelCathodeRearAxisY.commands.jogBackward,
                           intOut := "Unit1.Em6.HmiInterface".intCondition.Axis_29.Jog.intOut,
                           workInterlockOK => "Unit1.Em6.ControlNodes".cm.Interlock.mendrelCathodeRearAxisY.permit.jogBackward);
   "Unit1.Em6.ControlNodes".cmMendrelCathodeRearAxisY.commands.jogForward := NOT #TRUE AND "Unit1.Em6.ControlNodes".cm.Interlock.mendrelCathodeRearAxisY.permit.jogForward;
   "Unit1.Em6.ControlNodes".cmMendrelCathodeRearAxisY.commands.jogBackward := NOT #TRUE AND "Unit1.Em6.ControlNodes".cm.Interlock.mendrelCathodeRearAxisY.permit.jogBackward;
END_REGION

REGION Network 217: CmMendrelCathodeRearAxisY Position Absolute Position0
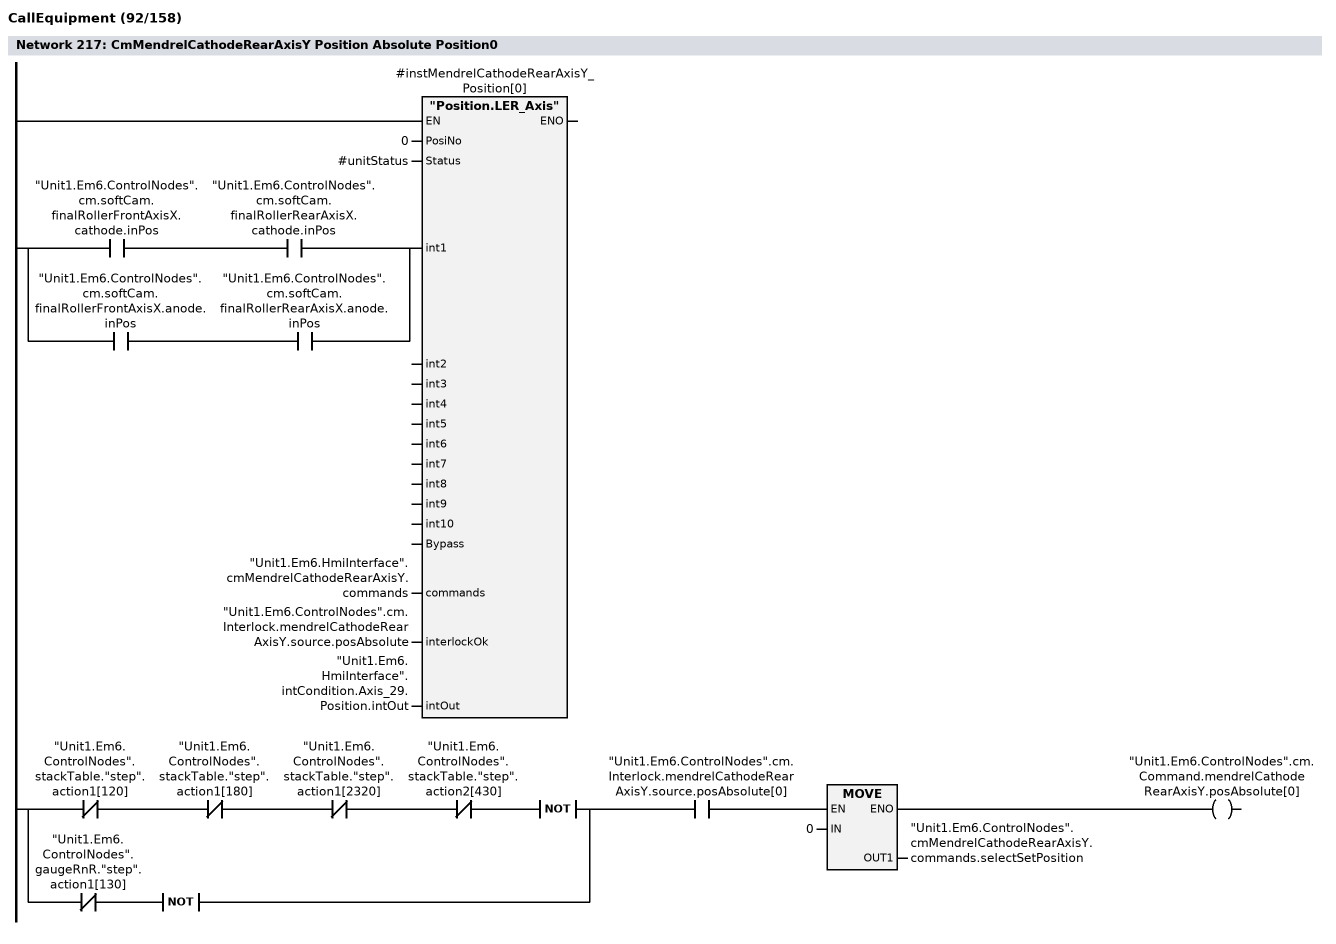
   RUNG wire#powerrail
      #instMendrelCathodeRearAxisY_Position[0](int1 := wire#w1, PosiNo := 0, Status := #unitStatus, int2 :=, int3 :=, int4 :=, int5 :=, int6 :=, int7 :=, int8 :=, int9 :=, int10 :=, Bypass :=, commands := "Unit1.Em6.HmiInterface".cmMendrelCathodeRearAxisY.commands, interlockOk := "Unit1.Em6.ControlNodes".cm.Interlock.mendrelCathodeRearAxisY.source.posAbsolute, intOut := "Unit1.Em6.HmiInterface".intCondition.Axis_29.Position.intOut)
   END_RUNG
   RUNG wire#powerrail
      Contact( "Unit1.Em6.ControlNodes".cm.softCam.finalRollerFrontAxisX.cathode.inPos )
      Contact( "Unit1.Em6.ControlNodes".cm.softCam.finalRollerRearAxisX.cathode.inPos )
   END_RUNG wire#w1
   RUNG wire#powerrail
      Contact( "Unit1.Em6.ControlNodes".cm.softCam.finalRollerFrontAxisX.anode.inPos )
      Contact( "Unit1.Em6.ControlNodes".cm.softCam.finalRollerRearAxisX.anode.inPos )
   END_RUNG wire#w1
   RUNG wire#powerrail
      I_Contact( "Unit1.Em6.ControlNodes".stackTable."step".action1[120] )
      I_Contact( "Unit1.Em6.ControlNodes".stackTable."step".action1[180] )
      I_Contact( "Unit1.Em6.ControlNodes".stackTable."step".action1[2320] )
      I_Contact( "Unit1.Em6.ControlNodes".stackTable."step".action2[430] )
      Not()
      wire#w2
      Contact( "Unit1.Em6.ControlNodes".cm.Interlock.mendrelCathodeRearAxisY.source.posAbsolute[0] )
      Move(in := 0, out1 => "Unit1.Em6.ControlNodes".cmMendrelCathodeRearAxisY.commands.selectSetPosition)
      Coil( "Unit1.Em6.ControlNodes".cm.Command.mendrelCathodeRearAxisY.posAbsolute[0] )
   END_RUNG
   RUNG wire#powerrail
      I_Contact( "Unit1.Em6.ControlNodes".gaugeRnR."step".action1[130] )
      Not()
   END_RUNG wire#w2
   // the same network as SCL:
   #instMendrelCathodeRearAxisY_Position[0](PosiNo := 0,   // "Position.LER_Axis"
                           Status := #unitStatus,
                           int1 := ("Unit1.Em6.ControlNodes".cm.softCam.finalRollerFrontAxisX.cathode.inPos AND "Unit1.Em6.ControlNodes".cm.softCam.finalRollerRearAxisX.cathode.inPos) OR ("Unit1.Em6.ControlNodes".cm.softCam.finalRollerFrontAxisX.anode.inPos AND "Unit1.Em6.ControlNodes".cm.softCam.finalRollerRearAxisX.anode.inPos),
                           commands := "Unit1.Em6.HmiInterface".cmMendrelCathodeRearAxisY.commands,
                           interlockOk := "Unit1.Em6.ControlNodes".cm.Interlock.mendrelCathodeRearAxisY.source.posAbsolute,
                           intOut := "Unit1.Em6.HmiInterface".intCondition.Axis_29.Position.intOut);
   #_w1 := (NOT (NOT "Unit1.Em6.ControlNodes".stackTable."step".action1[120] AND NOT "Unit1.Em6.ControlNodes".stackTable."step".action1[180] AND NOT "Unit1.Em6.ControlNodes".stackTable."step".action1[2320] AND NOT "Unit1.Em6.ControlNodes".stackTable."step".action2[430]) OR NOT (NOT "Unit1.Em6.ControlNodes".gaugeRnR."step".action1[130])) AND "Unit1.Em6.ControlNodes".cm.Interlock.mendrelCathodeRearAxisY.source.posAbsolute[0];
   IF #_w1 THEN "Unit1.Em6.ControlNodes".cmMendrelCathodeRearAxisY.commands.selectSetPosition := 0; END_IF;
   "Unit1.Em6.ControlNodes".cm.Command.mendrelCathodeRearAxisY.posAbsolute[0] := #_w1;
END_REGION

REGION Network 218: CmMendrelCathodeRearAxisY Position Absolute Position1
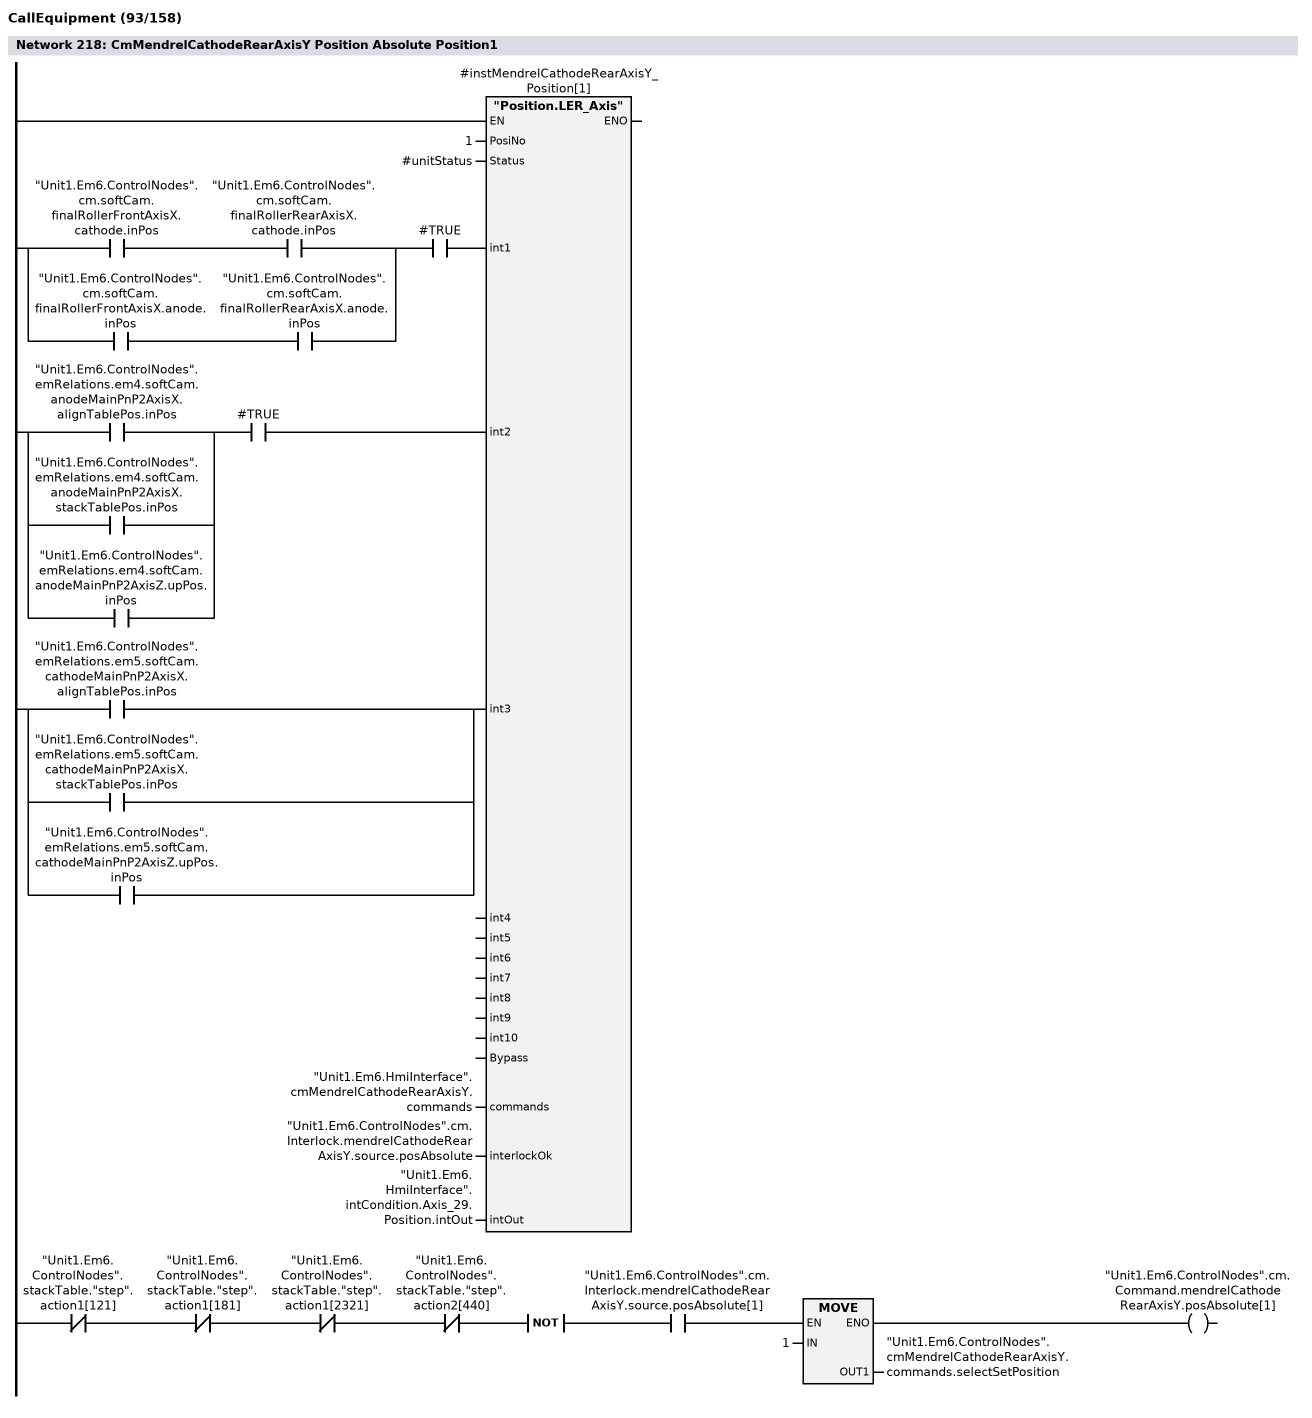
   RUNG wire#powerrail
      #instMendrelCathodeRearAxisY_Position[1](int1 := wire#w2, int2 := wire#w4, int3 := wire#w5, PosiNo := 1, Status := #unitStatus, int4 :=, int5 :=, int6 :=, int7 :=, int8 :=, int9 :=, int10 :=, Bypass :=, commands := "Unit1.Em6.HmiInterface".cmMendrelCathodeRearAxisY.commands, interlockOk := "Unit1.Em6.ControlNodes".cm.Interlock.mendrelCathodeRearAxisY.source.posAbsolute, intOut := "Unit1.Em6.HmiInterface".intCondition.Axis_29.Position.intOut)
   END_RUNG
   RUNG wire#powerrail
      Contact( "Unit1.Em6.ControlNodes".cm.softCam.finalRollerFrontAxisX.cathode.inPos )
      Contact( "Unit1.Em6.ControlNodes".cm.softCam.finalRollerRearAxisX.cathode.inPos )
      wire#w1
      Contact( #TRUE )
   END_RUNG wire#w2
   RUNG wire#powerrail
      Contact( "Unit1.Em6.ControlNodes".cm.softCam.finalRollerFrontAxisX.anode.inPos )
      Contact( "Unit1.Em6.ControlNodes".cm.softCam.finalRollerRearAxisX.anode.inPos )
   END_RUNG wire#w1
   RUNG wire#powerrail
      Contact( "Unit1.Em6.ControlNodes".emRelations.em4.softCam.anodeMainPnP2AxisX.alignTablePos.inPos )
      wire#w3
      Contact( #TRUE )
   END_RUNG wire#w4
   RUNG wire#powerrail
      Contact( "Unit1.Em6.ControlNodes".emRelations.em4.softCam.anodeMainPnP2AxisX.stackTablePos.inPos )
   END_RUNG wire#w3
   RUNG wire#powerrail
      Contact( "Unit1.Em6.ControlNodes".emRelations.em4.softCam.anodeMainPnP2AxisZ.upPos.inPos )
   END_RUNG wire#w3
   RUNG wire#powerrail
      Contact( "Unit1.Em6.ControlNodes".emRelations.em5.softCam.cathodeMainPnP2AxisX.alignTablePos.inPos )
   END_RUNG wire#w5
   RUNG wire#powerrail
      Contact( "Unit1.Em6.ControlNodes".emRelations.em5.softCam.cathodeMainPnP2AxisX.stackTablePos.inPos )
   END_RUNG wire#w5
   RUNG wire#powerrail
      Contact( "Unit1.Em6.ControlNodes".emRelations.em5.softCam.cathodeMainPnP2AxisZ.upPos.inPos )
   END_RUNG wire#w5
   RUNG wire#powerrail
      I_Contact( "Unit1.Em6.ControlNodes".stackTable."step".action1[121] )
      I_Contact( "Unit1.Em6.ControlNodes".stackTable."step".action1[181] )
      I_Contact( "Unit1.Em6.ControlNodes".stackTable."step".action1[2321] )
      I_Contact( "Unit1.Em6.ControlNodes".stackTable."step".action2[440] )
      Not()
      Contact( "Unit1.Em6.ControlNodes".cm.Interlock.mendrelCathodeRearAxisY.source.posAbsolute[1] )
      Move(in := 1, out1 => "Unit1.Em6.ControlNodes".cmMendrelCathodeRearAxisY.commands.selectSetPosition)
      Coil( "Unit1.Em6.ControlNodes".cm.Command.mendrelCathodeRearAxisY.posAbsolute[1] )
   END_RUNG
   // the same network as SCL:
   #instMendrelCathodeRearAxisY_Position[1](PosiNo := 1,   // "Position.LER_Axis"
                           Status := #unitStatus,
                           int1 := (("Unit1.Em6.ControlNodes".cm.softCam.finalRollerFrontAxisX.cathode.inPos AND "Unit1.Em6.ControlNodes".cm.softCam.finalRollerRearAxisX.cathode.inPos) OR ("Unit1.Em6.ControlNodes".cm.softCam.finalRollerFrontAxisX.anode.inPos AND "Unit1.Em6.ControlNodes".cm.softCam.finalRollerRearAxisX.anode.inPos)) AND #TRUE,
                           int2 := ("Unit1.Em6.ControlNodes".emRelations.em4.softCam.anodeMainPnP2AxisX.alignTablePos.inPos OR "Unit1.Em6.ControlNodes".emRelations.em4.softCam.anodeMainPnP2AxisX.stackTablePos.inPos OR "Unit1.Em6.ControlNodes".emRelations.em4.softCam.anodeMainPnP2AxisZ.upPos.inPos) AND #TRUE,
                           int3 := "Unit1.Em6.ControlNodes".emRelations.em5.softCam.cathodeMainPnP2AxisX.alignTablePos.inPos OR "Unit1.Em6.ControlNodes".emRelations.em5.softCam.cathodeMainPnP2AxisX.stackTablePos.inPos OR "Unit1.Em6.ControlNodes".emRelations.em5.softCam.cathodeMainPnP2AxisZ.upPos.inPos,
                           commands := "Unit1.Em6.HmiInterface".cmMendrelCathodeRearAxisY.commands,
                           interlockOk := "Unit1.Em6.ControlNodes".cm.Interlock.mendrelCathodeRearAxisY.source.posAbsolute,
                           intOut := "Unit1.Em6.HmiInterface".intCondition.Axis_29.Position.intOut);
   #_w1 := NOT (NOT "Unit1.Em6.ControlNodes".stackTable."step".action1[121] AND NOT "Unit1.Em6.ControlNodes".stackTable."step".action1[181] AND NOT "Unit1.Em6.ControlNodes".stackTable."step".action1[2321] AND NOT "Unit1.Em6.ControlNodes".stackTable."step".action2[440]) AND "Unit1.Em6.ControlNodes".cm.Interlock.mendrelCathodeRearAxisY.source.posAbsolute[1];
   IF #_w1 THEN "Unit1.Em6.ControlNodes".cmMendrelCathodeRearAxisY.commands.selectSetPosition := 1; END_IF;
   "Unit1.Em6.ControlNodes".cm.Command.mendrelCathodeRearAxisY.posAbsolute[1] := #_w1;
END_REGION

REGION Network 219: CmMendrelCathodeRearAxisY Position Absolute Position2
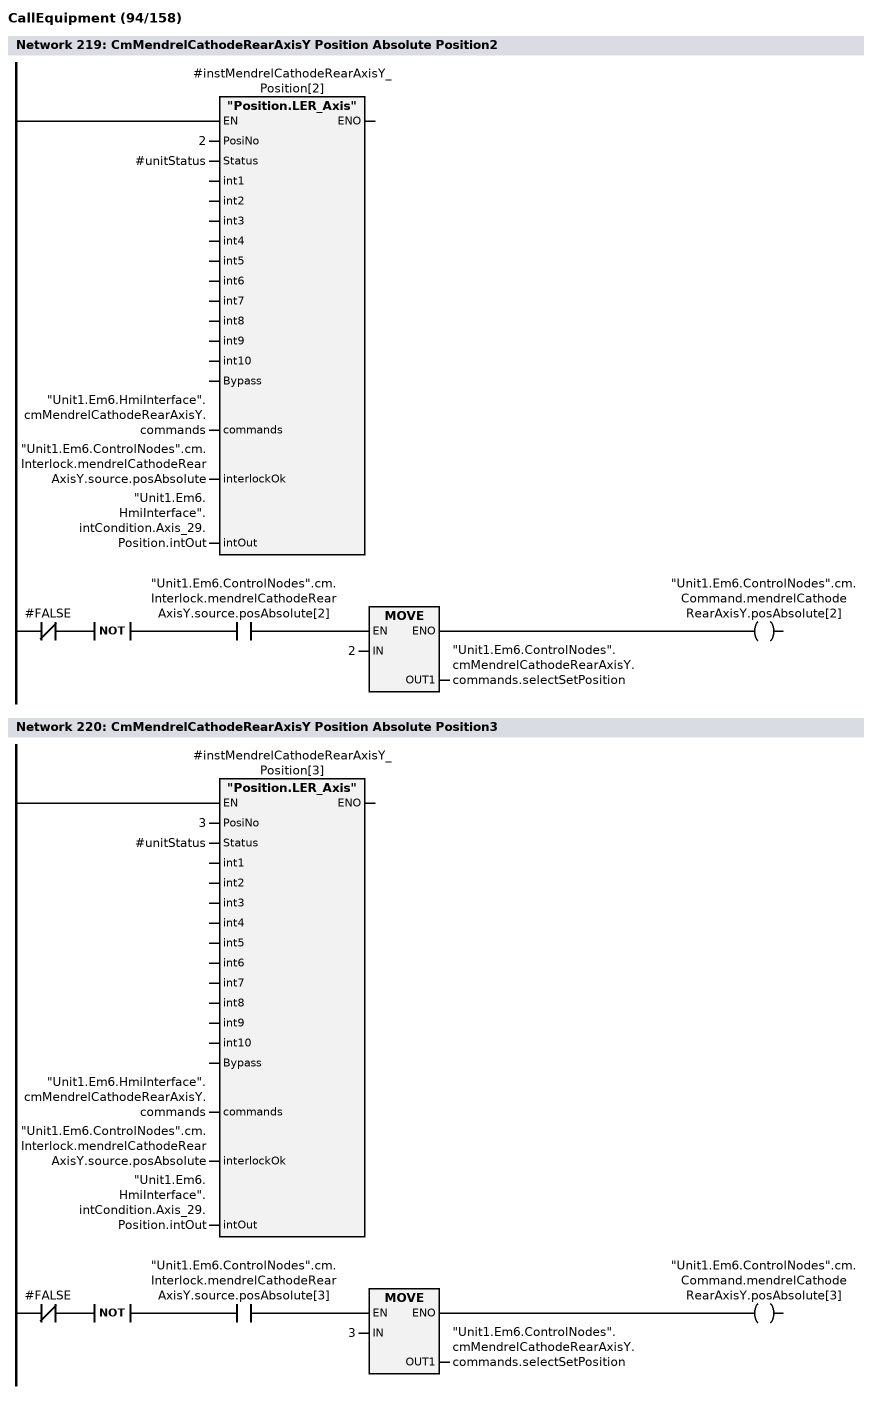
   RUNG wire#powerrail
      #instMendrelCathodeRearAxisY_Position[2](PosiNo := 2, Status := #unitStatus, int1 :=, int2 :=, int3 :=, int4 :=, int5 :=, int6 :=, int7 :=, int8 :=, int9 :=, int10 :=, Bypass :=, commands := "Unit1.Em6.HmiInterface".cmMendrelCathodeRearAxisY.commands, interlockOk := "Unit1.Em6.ControlNodes".cm.Interlock.mendrelCathodeRearAxisY.source.posAbsolute, intOut := "Unit1.Em6.HmiInterface".intCondition.Axis_29.Position.intOut)
   END_RUNG
   RUNG wire#powerrail
      I_Contact( #FALSE )
      Not()
      Contact( "Unit1.Em6.ControlNodes".cm.Interlock.mendrelCathodeRearAxisY.source.posAbsolute[2] )
      Move(in := 2, out1 => "Unit1.Em6.ControlNodes".cmMendrelCathodeRearAxisY.commands.selectSetPosition)
      Coil( "Unit1.Em6.ControlNodes".cm.Command.mendrelCathodeRearAxisY.posAbsolute[2] )
   END_RUNG
   // the same network as SCL:
   #instMendrelCathodeRearAxisY_Position[2](PosiNo := 2,   // "Position.LER_Axis"
                           Status := #unitStatus,
                           commands := "Unit1.Em6.HmiInterface".cmMendrelCathodeRearAxisY.commands,
                           interlockOk := "Unit1.Em6.ControlNodes".cm.Interlock.mendrelCathodeRearAxisY.source.posAbsolute,
                           intOut := "Unit1.Em6.HmiInterface".intCondition.Axis_29.Position.intOut);
   #_w1 := NOT (NOT #FALSE) AND "Unit1.Em6.ControlNodes".cm.Interlock.mendrelCathodeRearAxisY.source.posAbsolute[2];
   IF #_w1 THEN "Unit1.Em6.ControlNodes".cmMendrelCathodeRearAxisY.commands.selectSetPosition := 2; END_IF;
   "Unit1.Em6.ControlNodes".cm.Command.mendrelCathodeRearAxisY.posAbsolute[2] := #_w1;
END_REGION

REGION Network 220: CmMendrelCathodeRearAxisY Position Absolute Position3
   RUNG wire#powerrail
      #instMendrelCathodeRearAxisY_Position[3](PosiNo := 3, Status := #unitStatus, int1 :=, int2 :=, int3 :=, int4 :=, int5 :=, int6 :=, int7 :=, int8 :=, int9 :=, int10 :=, Bypass :=, commands := "Unit1.Em6.HmiInterface".cmMendrelCathodeRearAxisY.commands, interlockOk := "Unit1.Em6.ControlNodes".cm.Interlock.mendrelCathodeRearAxisY.source.posAbsolute, intOut := "Unit1.Em6.HmiInterface".intCondition.Axis_29.Position.intOut)
   END_RUNG
   RUNG wire#powerrail
      I_Contact( #FALSE )
      Not()
      Contact( "Unit1.Em6.ControlNodes".cm.Interlock.mendrelCathodeRearAxisY.source.posAbsolute[3] )
      Move(in := 3, out1 => "Unit1.Em6.ControlNodes".cmMendrelCathodeRearAxisY.commands.selectSetPosition)
      Coil( "Unit1.Em6.ControlNodes".cm.Command.mendrelCathodeRearAxisY.posAbsolute[3] )
   END_RUNG
   // the same network as SCL:
   #instMendrelCathodeRearAxisY_Position[3](PosiNo := 3,   // "Position.LER_Axis"
                           Status := #unitStatus,
                           commands := "Unit1.Em6.HmiInterface".cmMendrelCathodeRearAxisY.commands,
                           interlockOk := "Unit1.Em6.ControlNodes".cm.Interlock.mendrelCathodeRearAxisY.source.posAbsolute,
                           intOut := "Unit1.Em6.HmiInterface".intCondition.Axis_29.Position.intOut);
   #_w1 := NOT (NOT #FALSE) AND "Unit1.Em6.ControlNodes".cm.Interlock.mendrelCathodeRearAxisY.source.posAbsolute[3];
   IF #_w1 THEN "Unit1.Em6.ControlNodes".cmMendrelCathodeRearAxisY.commands.selectSetPosition := 3; END_IF;
   "Unit1.Em6.ControlNodes".cm.Command.mendrelCathodeRearAxisY.posAbsolute[3] := #_w1;
END_REGION

REGION Network 221: CmMendrelCathodeRearAxisY Position Absolute Position4
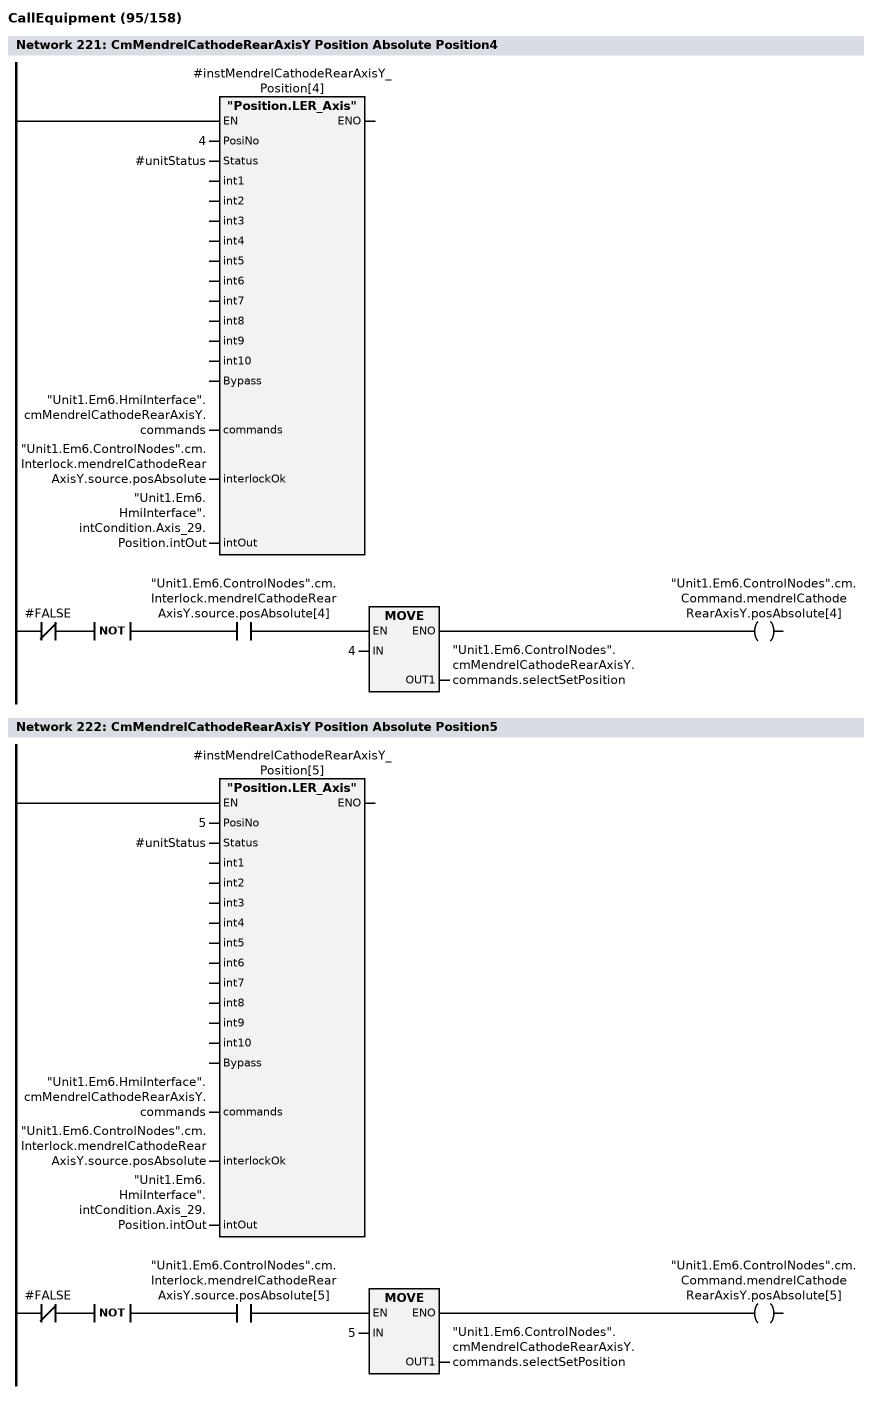
   RUNG wire#powerrail
      #instMendrelCathodeRearAxisY_Position[4](PosiNo := 4, Status := #unitStatus, int1 :=, int2 :=, int3 :=, int4 :=, int5 :=, int6 :=, int7 :=, int8 :=, int9 :=, int10 :=, Bypass :=, commands := "Unit1.Em6.HmiInterface".cmMendrelCathodeRearAxisY.commands, interlockOk := "Unit1.Em6.ControlNodes".cm.Interlock.mendrelCathodeRearAxisY.source.posAbsolute, intOut := "Unit1.Em6.HmiInterface".intCondition.Axis_29.Position.intOut)
   END_RUNG
   RUNG wire#powerrail
      I_Contact( #FALSE )
      Not()
      Contact( "Unit1.Em6.ControlNodes".cm.Interlock.mendrelCathodeRearAxisY.source.posAbsolute[4] )
      Move(in := 4, out1 => "Unit1.Em6.ControlNodes".cmMendrelCathodeRearAxisY.commands.selectSetPosition)
      Coil( "Unit1.Em6.ControlNodes".cm.Command.mendrelCathodeRearAxisY.posAbsolute[4] )
   END_RUNG
   // the same network as SCL:
   #instMendrelCathodeRearAxisY_Position[4](PosiNo := 4,   // "Position.LER_Axis"
                           Status := #unitStatus,
                           commands := "Unit1.Em6.HmiInterface".cmMendrelCathodeRearAxisY.commands,
                           interlockOk := "Unit1.Em6.ControlNodes".cm.Interlock.mendrelCathodeRearAxisY.source.posAbsolute,
                           intOut := "Unit1.Em6.HmiInterface".intCondition.Axis_29.Position.intOut);
   #_w1 := NOT (NOT #FALSE) AND "Unit1.Em6.ControlNodes".cm.Interlock.mendrelCathodeRearAxisY.source.posAbsolute[4];
   IF #_w1 THEN "Unit1.Em6.ControlNodes".cmMendrelCathodeRearAxisY.commands.selectSetPosition := 4; END_IF;
   "Unit1.Em6.ControlNodes".cm.Command.mendrelCathodeRearAxisY.posAbsolute[4] := #_w1;
END_REGION

REGION Network 222: CmMendrelCathodeRearAxisY Position Absolute Position5
   RUNG wire#powerrail
      #instMendrelCathodeRearAxisY_Position[5](PosiNo := 5, Status := #unitStatus, int1 :=, int2 :=, int3 :=, int4 :=, int5 :=, int6 :=, int7 :=, int8 :=, int9 :=, int10 :=, Bypass :=, commands := "Unit1.Em6.HmiInterface".cmMendrelCathodeRearAxisY.commands, interlockOk := "Unit1.Em6.ControlNodes".cm.Interlock.mendrelCathodeRearAxisY.source.posAbsolute, intOut := "Unit1.Em6.HmiInterface".intCondition.Axis_29.Position.intOut)
   END_RUNG
   RUNG wire#powerrail
      I_Contact( #FALSE )
      Not()
      Contact( "Unit1.Em6.ControlNodes".cm.Interlock.mendrelCathodeRearAxisY.source.posAbsolute[5] )
      Move(in := 5, out1 => "Unit1.Em6.ControlNodes".cmMendrelCathodeRearAxisY.commands.selectSetPosition)
      Coil( "Unit1.Em6.ControlNodes".cm.Command.mendrelCathodeRearAxisY.posAbsolute[5] )
   END_RUNG
   // the same network as SCL:
   #instMendrelCathodeRearAxisY_Position[5](PosiNo := 5,   // "Position.LER_Axis"
                           Status := #unitStatus,
                           commands := "Unit1.Em6.HmiInterface".cmMendrelCathodeRearAxisY.commands,
                           interlockOk := "Unit1.Em6.ControlNodes".cm.Interlock.mendrelCathodeRearAxisY.source.posAbsolute,
                           intOut := "Unit1.Em6.HmiInterface".intCondition.Axis_29.Position.intOut);
   #_w1 := NOT (NOT #FALSE) AND "Unit1.Em6.ControlNodes".cm.Interlock.mendrelCathodeRearAxisY.source.posAbsolute[5];
   IF #_w1 THEN "Unit1.Em6.ControlNodes".cmMendrelCathodeRearAxisY.commands.selectSetPosition := 5; END_IF;
   "Unit1.Em6.ControlNodes".cm.Command.mendrelCathodeRearAxisY.posAbsolute[5] := #_w1;
END_REGION

REGION Network 223: CmMendrelCathodeRearAxisY Summary Command
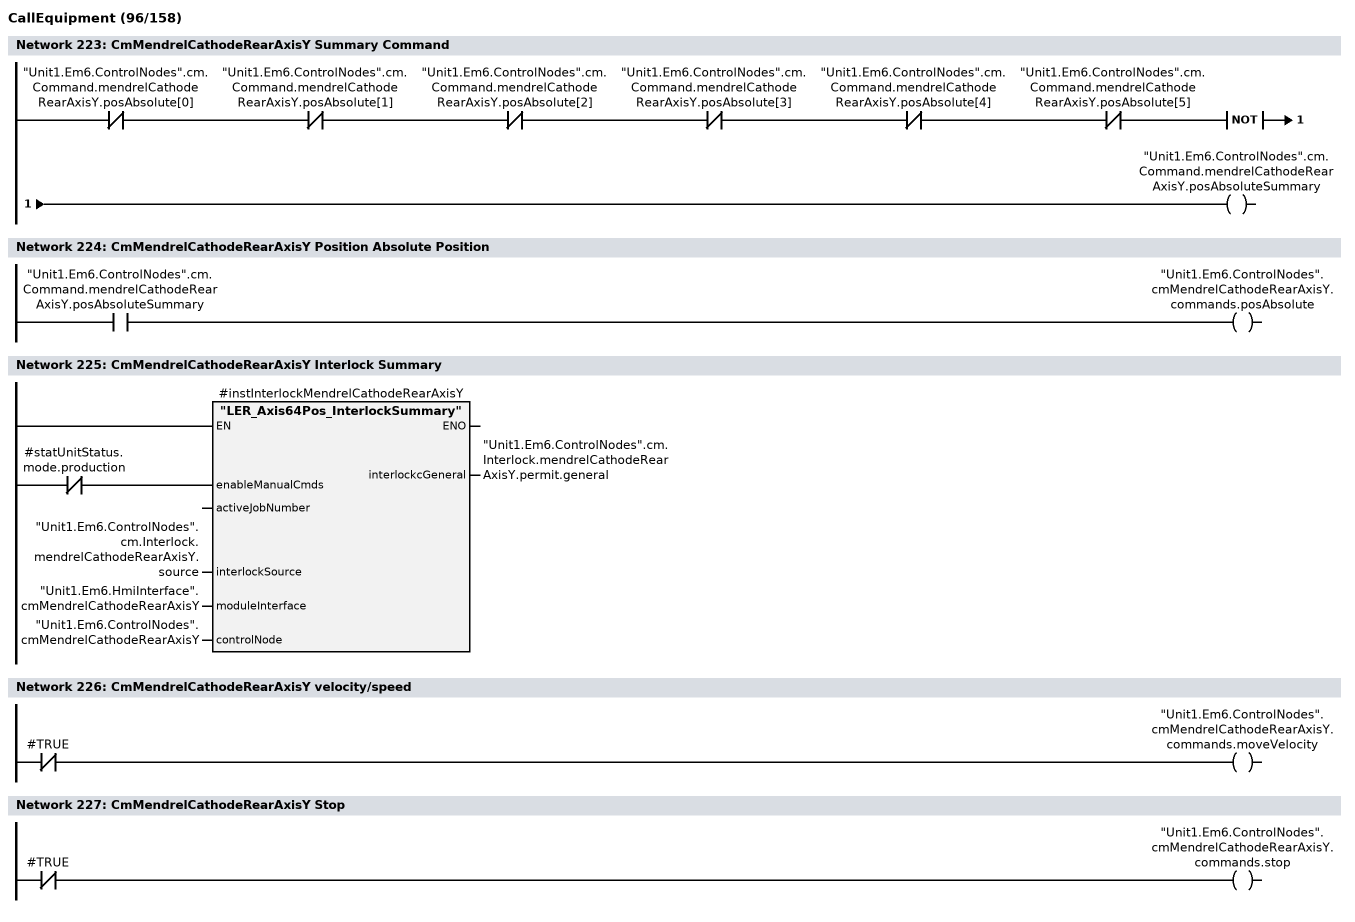
   RUNG wire#powerrail
      I_Contact( "Unit1.Em6.ControlNodes".cm.Command.mendrelCathodeRearAxisY.posAbsolute[0] )
      I_Contact( "Unit1.Em6.ControlNodes".cm.Command.mendrelCathodeRearAxisY.posAbsolute[1] )
      I_Contact( "Unit1.Em6.ControlNodes".cm.Command.mendrelCathodeRearAxisY.posAbsolute[2] )
      I_Contact( "Unit1.Em6.ControlNodes".cm.Command.mendrelCathodeRearAxisY.posAbsolute[3] )
      I_Contact( "Unit1.Em6.ControlNodes".cm.Command.mendrelCathodeRearAxisY.posAbsolute[4] )
      I_Contact( "Unit1.Em6.ControlNodes".cm.Command.mendrelCathodeRearAxisY.posAbsolute[5] )
      Not()
      Coil( "Unit1.Em6.ControlNodes".cm.Command.mendrelCathodeRearAxisY.posAbsoluteSummary )
   END_RUNG
   // the same network as SCL:
   "Unit1.Em6.ControlNodes".cm.Command.mendrelCathodeRearAxisY.posAbsoluteSummary := NOT (NOT "Unit1.Em6.ControlNodes".cm.Command.mendrelCathodeRearAxisY.posAbsolute[0] AND NOT "Unit1.Em6.ControlNodes".cm.Command.mendrelCathodeRearAxisY.posAbsolute[1] AND NOT "Unit1.Em6.ControlNodes".cm.Command.mendrelCathodeRearAxisY.posAbsolute[2] AND NOT "Unit1.Em6.ControlNodes".cm.Command.mendrelCathodeRearAxisY.posAbsolute[3] AND NOT "Unit1.Em6.ControlNodes".cm.Command.mendrelCathodeRearAxisY.posAbsolute[4] AND NOT "Unit1.Em6.ControlNodes".cm.Command.mendrelCathodeRearAxisY.posAbsolute[5]);
END_REGION

REGION Network 224: CmMendrelCathodeRearAxisY Position Absolute Position
   RUNG wire#powerrail
      Contact( "Unit1.Em6.ControlNodes".cm.Command.mendrelCathodeRearAxisY.posAbsoluteSummary )
      Coil( "Unit1.Em6.ControlNodes".cmMendrelCathodeRearAxisY.commands.posAbsolute )
   END_RUNG
   // the same network as SCL:
   "Unit1.Em6.ControlNodes".cmMendrelCathodeRearAxisY.commands.posAbsolute := "Unit1.Em6.ControlNodes".cm.Command.mendrelCathodeRearAxisY.posAbsoluteSummary;
END_REGION

REGION Network 225: CmMendrelCathodeRearAxisY Interlock Summary
   RUNG wire#powerrail
      #instInterlockMendrelCathodeRearAxisY(enableManualCmds := wire#w1, activeJobNumber :=, interlockSource := "Unit1.Em6.ControlNodes".cm.Interlock.mendrelCathodeRearAxisY.source, moduleInterface := "Unit1.Em6.HmiInterface".cmMendrelCathodeRearAxisY, controlNode := "Unit1.Em6.ControlNodes".cmMendrelCathodeRearAxisY, interlockcGeneral => "Unit1.Em6.ControlNodes".cm.Interlock.mendrelCathodeRearAxisY.permit.general)
   END_RUNG
   RUNG wire#powerrail
      I_Contact( #statUnitStatus.mode.production )
   END_RUNG wire#w1
   // the same network as SCL:
   #instInterlockMendrelCathodeRearAxisY(enableManualCmds := NOT #statUnitStatus.mode.production,   // "LER_Axis64Pos_InterlockSummary"
                           interlockSource := "Unit1.Em6.ControlNodes".cm.Interlock.mendrelCathodeRearAxisY.source,
                           moduleInterface := "Unit1.Em6.HmiInterface".cmMendrelCathodeRearAxisY,
                           controlNode := "Unit1.Em6.ControlNodes".cmMendrelCathodeRearAxisY,
                           interlockcGeneral => "Unit1.Em6.ControlNodes".cm.Interlock.mendrelCathodeRearAxisY.permit.general);
END_REGION

REGION Network 226: CmMendrelCathodeRearAxisY velocity/speed
   RUNG wire#powerrail
      I_Contact( #TRUE )
      Coil( "Unit1.Em6.ControlNodes".cmMendrelCathodeRearAxisY.commands.moveVelocity )
   END_RUNG
   // the same network as SCL:
   "Unit1.Em6.ControlNodes".cmMendrelCathodeRearAxisY.commands.moveVelocity := NOT #TRUE;
END_REGION

REGION Network 227: CmMendrelCathodeRearAxisY Stop
   RUNG wire#powerrail
      I_Contact( #TRUE )
      Coil( "Unit1.Em6.ControlNodes".cmMendrelCathodeRearAxisY.commands.stop )
   END_RUNG
   // the same network as SCL:
   "Unit1.Em6.ControlNodes".cmMendrelCathodeRearAxisY.commands.stop := NOT #TRUE;
END_REGION

REGION Network 228: Call CM Cathode Mandrel Rear Y-Axis (LBC_Axis64Pos)
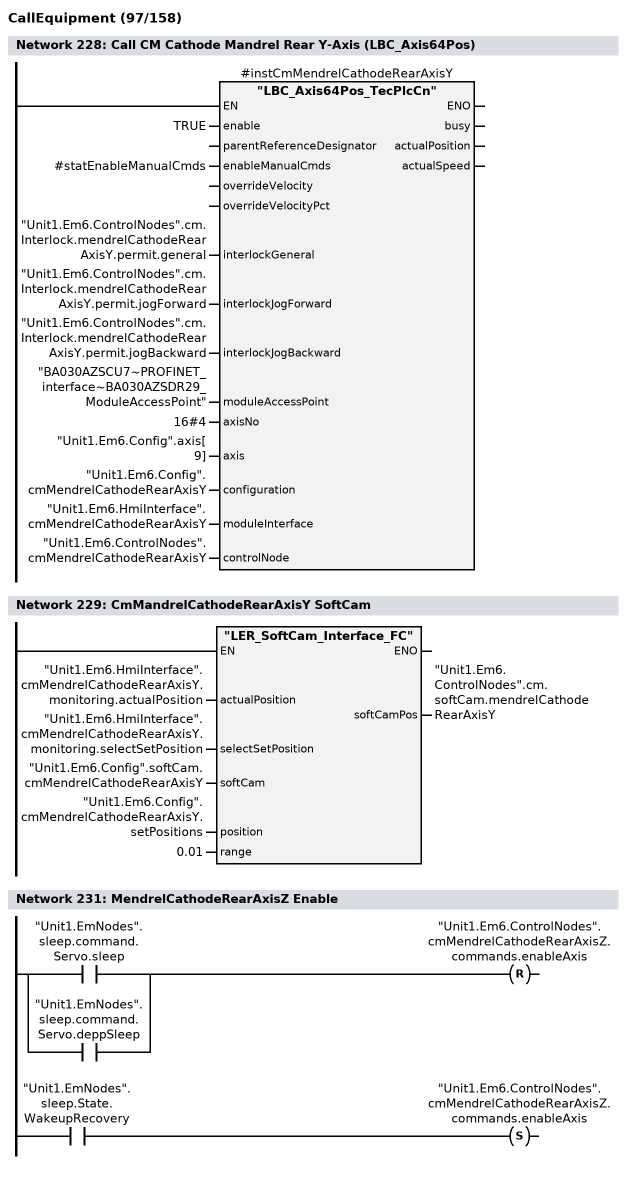
   RUNG wire#powerrail
      #instCmMendrelCathodeRearAxisY(enable := TRUE, parentReferenceDesignator :=, enableManualCmds := #statEnableManualCmds, overrideVelocity :=, overrideVelocityPct :=, interlockGeneral := "Unit1.Em6.ControlNodes".cm.Interlock.mendrelCathodeRearAxisY.permit.general, interlockJogForward := "Unit1.Em6.ControlNodes".cm.Interlock.mendrelCathodeRearAxisY.permit.jogForward, interlockJogBackward := "Unit1.Em6.ControlNodes".cm.Interlock.mendrelCathodeRearAxisY.permit.jogBackward, moduleAccessPoint := "BA030AZSCU7~PROFINET_interface~BA030AZSDR29_ModuleAccessPoint", axisNo := 16#4, axis := "Unit1.Em6.Config".axis[9], configuration := "Unit1.Em6.Config".cmMendrelCathodeRearAxisY, moduleInterface := "Unit1.Em6.HmiInterface".cmMendrelCathodeRearAxisY, controlNode := "Unit1.Em6.ControlNodes".cmMendrelCathodeRearAxisY, busy =>, actualPosition =>, actualSpeed =>)
   END_RUNG
   // the same network as SCL:
   #instCmMendrelCathodeRearAxisY(enable := TRUE,   // "LBC_Axis64Pos_TecPlcCn"
                           enableManualCmds := #statEnableManualCmds,
                           interlockGeneral := "Unit1.Em6.ControlNodes".cm.Interlock.mendrelCathodeRearAxisY.permit.general,
                           interlockJogForward := "Unit1.Em6.ControlNodes".cm.Interlock.mendrelCathodeRearAxisY.permit.jogForward,
                           interlockJogBackward := "Unit1.Em6.ControlNodes".cm.Interlock.mendrelCathodeRearAxisY.permit.jogBackward,
                           moduleAccessPoint := "BA030AZSCU7~PROFINET_interface~BA030AZSDR29_ModuleAccessPoint",
                           axisNo := 16#4,
                           axis := "Unit1.Em6.Config".axis[9],
                           configuration := "Unit1.Em6.Config".cmMendrelCathodeRearAxisY,
                           moduleInterface := "Unit1.Em6.HmiInterface".cmMendrelCathodeRearAxisY,
                           controlNode := "Unit1.Em6.ControlNodes".cmMendrelCathodeRearAxisY);
END_REGION

REGION Network 229: CmMandrelCathodeRearAxisY SoftCam
   RUNG wire#powerrail
      "LER_SoftCam_Interface_FC"(actualPosition := "Unit1.Em6.HmiInterface".cmMendrelCathodeRearAxisY.monitoring.actualPosition, selectSetPosition := "Unit1.Em6.HmiInterface".cmMendrelCathodeRearAxisY.monitoring.selectSetPosition, softCam := "Unit1.Em6.Config".softCam.cmMendrelCathodeRearAxisY, position := "Unit1.Em6.Config".cmMendrelCathodeRearAxisY.setPositions, range := 0.01, softCamPos => "Unit1.Em6.ControlNodes".cm.softCam.mendrelCathodeRearAxisY)
   END_RUNG
   // the same network as SCL:
   "LER_SoftCam_Interface_FC"(actualPosition := "Unit1.Em6.HmiInterface".cmMendrelCathodeRearAxisY.monitoring.actualPosition,
                           selectSetPosition := "Unit1.Em6.HmiInterface".cmMendrelCathodeRearAxisY.monitoring.selectSetPosition,
                           softCam := "Unit1.Em6.Config".softCam.cmMendrelCathodeRearAxisY,
                           position := "Unit1.Em6.Config".cmMendrelCathodeRearAxisY.setPositions,
                           range := 0.01,
                           softCamPos => "Unit1.Em6.ControlNodes".cm.softCam.mendrelCathodeRearAxisY);
END_REGION

REGION Network 231: MendrelCathodeRearAxisZ Enable
   RUNG wire#powerrail
      Contact( "Unit1.EmNodes".sleep.command.Servo.sleep )
      wire#w1
      R_Coil( "Unit1.Em6.ControlNodes".cmMendrelCathodeRearAxisZ.commands.enableAxis )
   END_RUNG
   RUNG wire#powerrail
      Contact( "Unit1.EmNodes".sleep.command.Servo.deppSleep )
   END_RUNG wire#w1
   RUNG wire#powerrail
      Contact( "Unit1.EmNodes".sleep.State.WakeupRecovery )
      S_Coil( "Unit1.Em6.ControlNodes".cmMendrelCathodeRearAxisZ.commands.enableAxis )
   END_RUNG
   // the same network as SCL:
   IF "Unit1.EmNodes".sleep.command.Servo.sleep OR "Unit1.EmNodes".sleep.command.Servo.deppSleep THEN
       "Unit1.Em6.ControlNodes".cmMendrelCathodeRearAxisZ.commands.enableAxis := FALSE;
   END_IF;
   IF "Unit1.EmNodes".sleep.State.WakeupRecovery THEN
       "Unit1.Em6.ControlNodes".cmMendrelCathodeRearAxisZ.commands.enableAxis := TRUE;
   END_IF;
END_REGION

REGION Network 232: CmmendrelCathodeRearAxisZ Home
